// TIA Portal V17 export
// export: Created 2025-04-22T12:08:34.2045134Z, ExportSetting WithDefaults, DisplayName Totally Integrated Automation Portal, DisplayVersion V17 Update 8, DisplayName TIA Portal Openness, DisplayVersion V17 Update 8, DisplayName TIA Portal Version Control Interface, DisplayVersion V17, DisplayName SINAMICS Startdrive Advanced, DisplayVersion V17 SP2, DisplayName SINAMICS Startdrive G110M, G120, G120C, G120D, G120P, G115D, DisplayVersion V17 SP2, DisplayName SINAMICS Startdrive G130, G150, S120, S150, SINAMICS MV, S210, DisplayVersion V17 SP2, DisplayName STEP 7 Professional, DisplayVersion V17 Update 8, DisplayName SINUMERIK ONE STEP 7 Toolbox, DisplayVersion V17 Update 12, DisplayName SINUMERIK 840D sl STEP 7 Toolbox, DisplayVersion V17 Update 12, DisplayName STEP 7 Safety, DisplayVersion V17 Update 6, DisplayName WinCC Advanced / Unified PC, DisplayVersion V17 Update 8
FUNCTION "FC2401_DBBS_CLADDING" : Void   // FC2401, LAD
TITLE = NCK Inputs
{ S7_Optimized_Access := 'FALSE' }
AUTHOR : ETXETAR
VERSION : 1.0
// stored: AutoNumber false, IsIECCheckEnabled false, SetENOAutomatically false, UDAEnableTagReadback false
   VAR_TEMP
      ERROR : Bool;   // ERROR
      ERROR_CODE : Int;   // ERROR CODE
      F1_RESET_SEMI_WORKS : Bool;   // FIXTURE 1 RESET SEMI WORKS
      F2_RESET_SEMI_WORKS : Bool;   // FIXTURE 2 RESET SEMI WORKS
      RESET_UGUD : Bool;   // RESET UGUD
      TAG_ERROR_01R : Int;   // TAG ERROR 01R
      TAG_ERROR_01L : Int;   // TAG ERROR 01L
   END_VAR
   VAR CONSTANT
      READ : Byte := 16#3;
      WRITE : Byte := 16#4;
   END_VAR
BEGIN

REGION Network 1: MACHINE CNC CYCLE UNIT 01 TRANSFER CHANNEL 1 - $A_DBB[0] / CYCLE SELECTION 01R
   // 0 --> NA
   // 1 --> PART CYCLE 01R
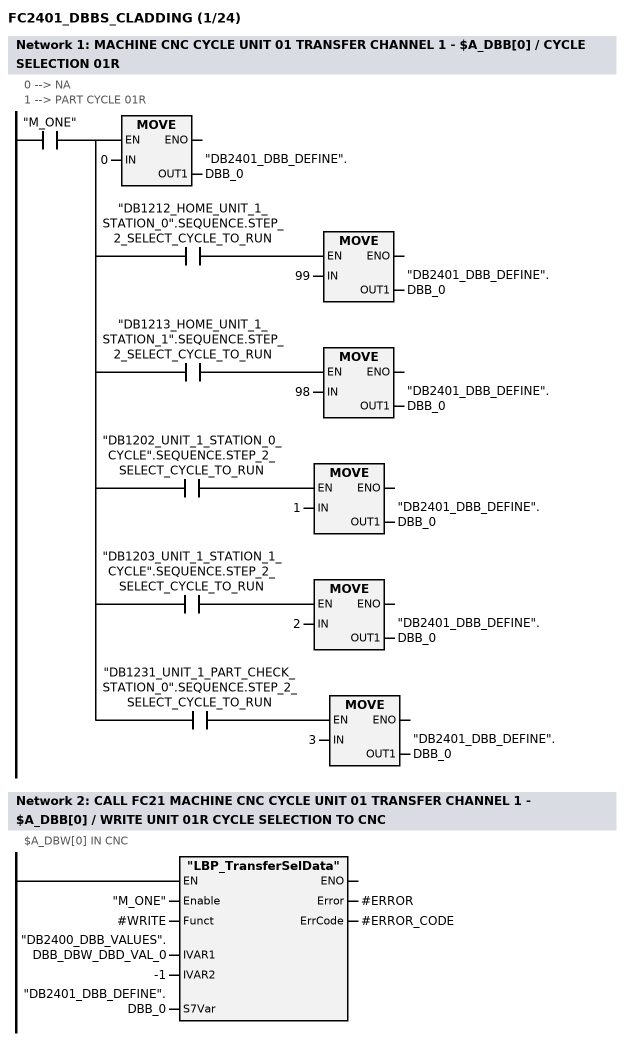
   RUNG wire#powerrail
      Contact( "M_ONE" )
      wire#w1
      { S7_GenerateENO := "TRUE" } Move(in := 0, out1 => "DB2401_DBB_DEFINE".DBB_0)
   END_RUNG
   RUNG wire#w1
      Contact( "DB1212_HOME_UNIT_1_STATION_0".SEQUENCE.STEP_2_SELECT_CYCLE_TO_RUN )
      { S7_GenerateENO := "TRUE" } Move(in := 99, out1 => "DB2401_DBB_DEFINE".DBB_0)
   END_RUNG
   RUNG wire#w1
      Contact( "DB1213_HOME_UNIT_1_STATION_1".SEQUENCE.STEP_2_SELECT_CYCLE_TO_RUN )
      { S7_GenerateENO := "TRUE" } Move(in := 98, out1 => "DB2401_DBB_DEFINE".DBB_0)
   END_RUNG
   RUNG wire#w1
      Contact( "DB1202_UNIT_1_STATION_0_CYCLE".SEQUENCE.STEP_2_SELECT_CYCLE_TO_RUN )
      { S7_GenerateENO := "TRUE" } Move(in := 1, out1 => "DB2401_DBB_DEFINE".DBB_0)
   END_RUNG
   RUNG wire#w1
      Contact( "DB1203_UNIT_1_STATION_1_CYCLE".SEQUENCE.STEP_2_SELECT_CYCLE_TO_RUN )
      { S7_GenerateENO := "TRUE" } Move(in := 2, out1 => "DB2401_DBB_DEFINE".DBB_0)
   END_RUNG
   RUNG wire#w1
      Contact( "DB1231_UNIT_1_PART_CHECK_STATION_0".SEQUENCE.STEP_2_SELECT_CYCLE_TO_RUN )
      { S7_GenerateENO := "TRUE" } Move(in := 3, out1 => "DB2401_DBB_DEFINE".DBB_0)
   END_RUNG
   // the same network as SCL:
   IF "M_ONE" THEN "DB2401_DBB_DEFINE".DBB_0 := 0; END_IF;
   IF "M_ONE" AND "DB1212_HOME_UNIT_1_STATION_0".SEQUENCE.STEP_2_SELECT_CYCLE_TO_RUN THEN
       "DB2401_DBB_DEFINE".DBB_0 := 99;
   END_IF;
   IF "M_ONE" AND "DB1213_HOME_UNIT_1_STATION_1".SEQUENCE.STEP_2_SELECT_CYCLE_TO_RUN THEN
       "DB2401_DBB_DEFINE".DBB_0 := 98;
   END_IF;
   IF "M_ONE" AND "DB1202_UNIT_1_STATION_0_CYCLE".SEQUENCE.STEP_2_SELECT_CYCLE_TO_RUN THEN
       "DB2401_DBB_DEFINE".DBB_0 := 1;
   END_IF;
   IF "M_ONE" AND "DB1203_UNIT_1_STATION_1_CYCLE".SEQUENCE.STEP_2_SELECT_CYCLE_TO_RUN THEN
       "DB2401_DBB_DEFINE".DBB_0 := 2;
   END_IF;
   IF "M_ONE" AND "DB1231_UNIT_1_PART_CHECK_STATION_0".SEQUENCE.STEP_2_SELECT_CYCLE_TO_RUN THEN
       "DB2401_DBB_DEFINE".DBB_0 := 3;
   END_IF;
END_REGION

REGION Network 2: CALL FC21 MACHINE CNC CYCLE UNIT 01 TRANSFER CHANNEL 1 - $A_DBB[0] / WRITE UNIT 01R CYCLE SELECTION TO CNC
   // $A_DBW[0] IN CNC
   RUNG wire#powerrail
      "LBP_TransferSelData"(Enable := "M_ONE", Funct := #WRITE, IVAR1 := "DB2400_DBB_VALUES".DBB_DBW_DBD_VAL_0, IVAR2 := -1, S7Var := "DB2401_DBB_DEFINE".DBB_0, Error => #ERROR, ErrCode => #ERROR_CODE)
   END_RUNG
   // the same network as SCL:
   "LBP_TransferSelData"(Enable := "M_ONE",
                         Funct := #WRITE,
                         IVAR1 := "DB2400_DBB_VALUES".DBB_DBW_DBD_VAL_0,
                         IVAR2 := -1,
                         S7Var := "DB2401_DBB_DEFINE".DBB_0,
                         Error => #ERROR,
                         ErrCode => #ERROR_CODE);
END_REGION

REGION Network 3: MACHINE CNC CYCLE UNIT 01 CLADDING CHANNEL 2 - $A_DBB[2] / CYCLE SELECTION PHD
   // 0 --> NA
   // 1 --> PHD CYCLE
   // 99 --> RETURN HOME CYCLE PHD
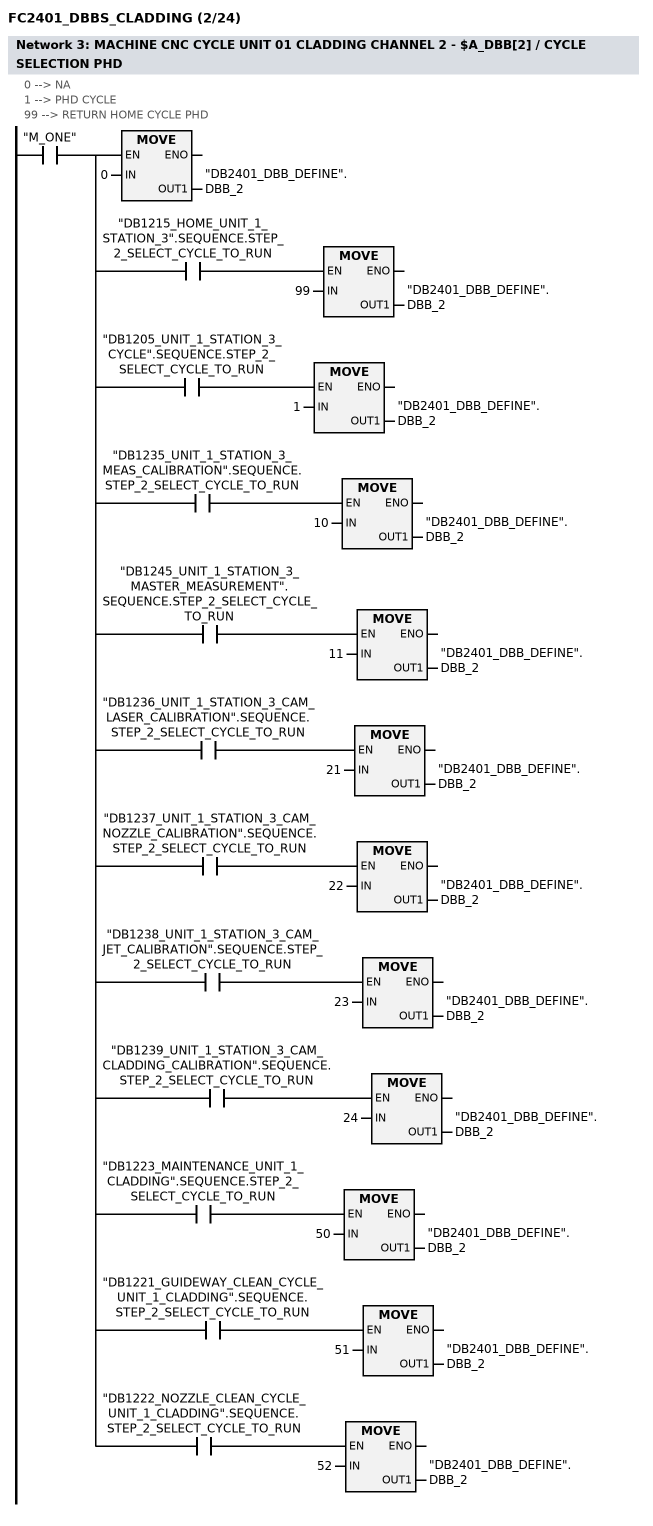
   RUNG wire#powerrail
      Contact( "M_ONE" )
      wire#w1
      { S7_GenerateENO := "TRUE" } Move(in := 0, out1 => "DB2401_DBB_DEFINE".DBB_2)
   END_RUNG
   RUNG wire#w1
      Contact( "DB1215_HOME_UNIT_1_STATION_3".SEQUENCE.STEP_2_SELECT_CYCLE_TO_RUN )
      { S7_GenerateENO := "TRUE" } Move(in := 99, out1 => "DB2401_DBB_DEFINE".DBB_2)
   END_RUNG
   RUNG wire#w1
      Contact( "DB1205_UNIT_1_STATION_3_CYCLE".SEQUENCE.STEP_2_SELECT_CYCLE_TO_RUN )
      { S7_GenerateENO := "TRUE" } Move(in := 1, out1 => "DB2401_DBB_DEFINE".DBB_2)
   END_RUNG
   RUNG wire#w1
      Contact( "DB1235_UNIT_1_STATION_3_MEAS_CALIBRATION".SEQUENCE.STEP_2_SELECT_CYCLE_TO_RUN )
      { S7_GenerateENO := "TRUE" } Move(in := 10, out1 => "DB2401_DBB_DEFINE".DBB_2)
   END_RUNG
   RUNG wire#w1
      Contact( "DB1245_UNIT_1_STATION_3_MASTER_MEASUREMENT".SEQUENCE.STEP_2_SELECT_CYCLE_TO_RUN )
      { S7_GenerateENO := "TRUE" } Move(in := 11, out1 => "DB2401_DBB_DEFINE".DBB_2)
   END_RUNG
   RUNG wire#w1
      Contact( "DB1236_UNIT_1_STATION_3_CAM_LASER_CALIBRATION".SEQUENCE.STEP_2_SELECT_CYCLE_TO_RUN )
      { S7_GenerateENO := "TRUE" } Move(in := 21, out1 => "DB2401_DBB_DEFINE".DBB_2)
   END_RUNG
   RUNG wire#w1
      Contact( "DB1237_UNIT_1_STATION_3_CAM_NOZZLE_CALIBRATION".SEQUENCE.STEP_2_SELECT_CYCLE_TO_RUN )
      { S7_GenerateENO := "TRUE" } Move(in := 22, out1 => "DB2401_DBB_DEFINE".DBB_2)
   END_RUNG
   RUNG wire#w1
      Contact( "DB1238_UNIT_1_STATION_3_CAM_JET_CALIBRATION".SEQUENCE.STEP_2_SELECT_CYCLE_TO_RUN )
      { S7_GenerateENO := "TRUE" } Move(in := 23, out1 => "DB2401_DBB_DEFINE".DBB_2)
   END_RUNG
   RUNG wire#w1
      Contact( "DB1239_UNIT_1_STATION_3_CAM_CLADDING_CALIBRATION".SEQUENCE.STEP_2_SELECT_CYCLE_TO_RUN )
      { S7_GenerateENO := "TRUE" } Move(in := 24, out1 => "DB2401_DBB_DEFINE".DBB_2)
   END_RUNG
   RUNG wire#w1
      Contact( "DB1223_MAINTENANCE_UNIT_1_CLADDING".SEQUENCE.STEP_2_SELECT_CYCLE_TO_RUN )
      { S7_GenerateENO := "TRUE" } Move(in := 50, out1 => "DB2401_DBB_DEFINE".DBB_2)
   END_RUNG
   RUNG wire#w1
      Contact( "DB1221_GUIDEWAY_CLEAN_CYCLE_UNIT_1_CLADDING".SEQUENCE.STEP_2_SELECT_CYCLE_TO_RUN )
      { S7_GenerateENO := "TRUE" } Move(in := 51, out1 => "DB2401_DBB_DEFINE".DBB_2)
   END_RUNG
   RUNG wire#w1
      Contact( "DB1222_NOZZLE_CLEAN_CYCLE_UNIT_1_CLADDING".SEQUENCE.STEP_2_SELECT_CYCLE_TO_RUN )
      { S7_GenerateENO := "TRUE" } Move(in := 52, out1 => "DB2401_DBB_DEFINE".DBB_2)
   END_RUNG
   // the same network as SCL:
   IF "M_ONE" THEN "DB2401_DBB_DEFINE".DBB_2 := 0; END_IF;
   IF "M_ONE" AND "DB1215_HOME_UNIT_1_STATION_3".SEQUENCE.STEP_2_SELECT_CYCLE_TO_RUN THEN
       "DB2401_DBB_DEFINE".DBB_2 := 99;
   END_IF;
   IF "M_ONE" AND "DB1205_UNIT_1_STATION_3_CYCLE".SEQUENCE.STEP_2_SELECT_CYCLE_TO_RUN THEN
       "DB2401_DBB_DEFINE".DBB_2 := 1;
   END_IF;
   IF "M_ONE" AND "DB1235_UNIT_1_STATION_3_MEAS_CALIBRATION".SEQUENCE.STEP_2_SELECT_CYCLE_TO_RUN THEN
       "DB2401_DBB_DEFINE".DBB_2 := 10;
   END_IF;
   IF "M_ONE" AND "DB1245_UNIT_1_STATION_3_MASTER_MEASUREMENT".SEQUENCE.STEP_2_SELECT_CYCLE_TO_RUN THEN
       "DB2401_DBB_DEFINE".DBB_2 := 11;
   END_IF;
   IF "M_ONE" AND "DB1236_UNIT_1_STATION_3_CAM_LASER_CALIBRATION".SEQUENCE.STEP_2_SELECT_CYCLE_TO_RUN THEN
       "DB2401_DBB_DEFINE".DBB_2 := 21;
   END_IF;
   IF "M_ONE" AND "DB1237_UNIT_1_STATION_3_CAM_NOZZLE_CALIBRATION".SEQUENCE.STEP_2_SELECT_CYCLE_TO_RUN THEN
       "DB2401_DBB_DEFINE".DBB_2 := 22;
   END_IF;
   IF "M_ONE" AND "DB1238_UNIT_1_STATION_3_CAM_JET_CALIBRATION".SEQUENCE.STEP_2_SELECT_CYCLE_TO_RUN THEN
       "DB2401_DBB_DEFINE".DBB_2 := 23;
   END_IF;
   IF "M_ONE" AND "DB1239_UNIT_1_STATION_3_CAM_CLADDING_CALIBRATION".SEQUENCE.STEP_2_SELECT_CYCLE_TO_RUN THEN
       "DB2401_DBB_DEFINE".DBB_2 := 24;
   END_IF;
   IF "M_ONE" AND "DB1223_MAINTENANCE_UNIT_1_CLADDING".SEQUENCE.STEP_2_SELECT_CYCLE_TO_RUN THEN
       "DB2401_DBB_DEFINE".DBB_2 := 50;
   END_IF;
   IF "M_ONE" AND "DB1221_GUIDEWAY_CLEAN_CYCLE_UNIT_1_CLADDING".SEQUENCE.STEP_2_SELECT_CYCLE_TO_RUN THEN
       "DB2401_DBB_DEFINE".DBB_2 := 51;
   END_IF;
   IF "M_ONE" AND "DB1222_NOZZLE_CLEAN_CYCLE_UNIT_1_CLADDING".SEQUENCE.STEP_2_SELECT_CYCLE_TO_RUN THEN
       "DB2401_DBB_DEFINE".DBB_2 := 52;
   END_IF;
END_REGION

REGION Network 4: CALL FC21 MACHINE CNC CYCLE UNIT 01 CLADDING CHANNEL 2 - $A_DBB[2] / WRITE UNIT 01R CYCLE SELECTION TO CNC
   // $A_DBW[0] IN CNC
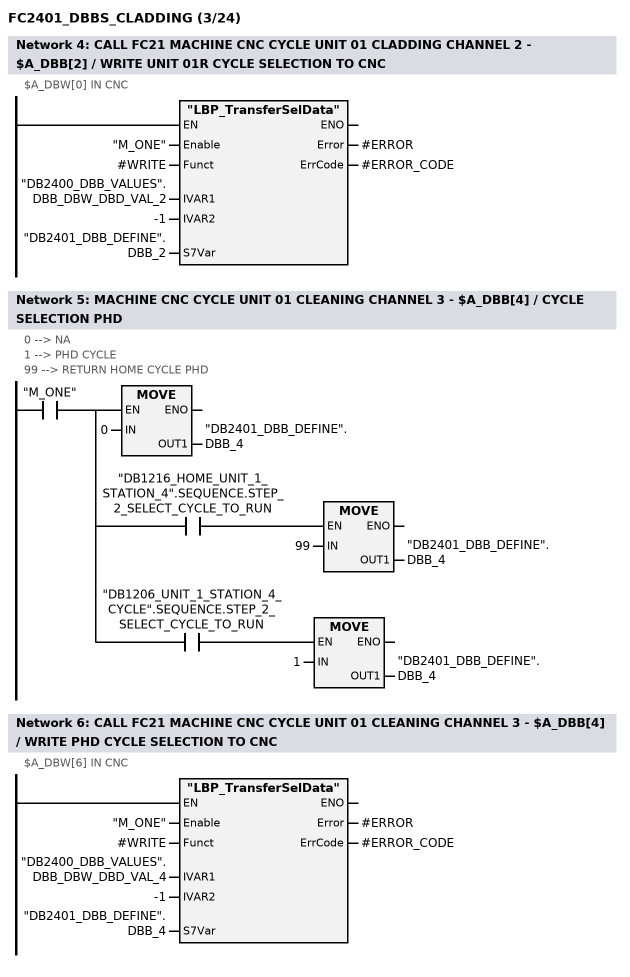
   RUNG wire#powerrail
      "LBP_TransferSelData"(Enable := "M_ONE", Funct := #WRITE, IVAR1 := "DB2400_DBB_VALUES".DBB_DBW_DBD_VAL_2, IVAR2 := -1, S7Var := "DB2401_DBB_DEFINE".DBB_2, Error => #ERROR, ErrCode => #ERROR_CODE)
   END_RUNG
   // the same network as SCL:
   "LBP_TransferSelData"(Enable := "M_ONE",
                         Funct := #WRITE,
                         IVAR1 := "DB2400_DBB_VALUES".DBB_DBW_DBD_VAL_2,
                         IVAR2 := -1,
                         S7Var := "DB2401_DBB_DEFINE".DBB_2,
                         Error => #ERROR,
                         ErrCode => #ERROR_CODE);
END_REGION

REGION Network 5: MACHINE CNC CYCLE UNIT 01 CLEANING CHANNEL 3 - $A_DBB[4] / CYCLE SELECTION PHD
   // 0 --> NA
   // 1 --> PHD CYCLE
   // 99 --> RETURN HOME CYCLE PHD
   RUNG wire#powerrail
      Contact( "M_ONE" )
      wire#w1
      { S7_GenerateENO := "TRUE" } Move(in := 0, out1 => "DB2401_DBB_DEFINE".DBB_4)
   END_RUNG
   RUNG wire#w1
      Contact( "DB1216_HOME_UNIT_1_STATION_4".SEQUENCE.STEP_2_SELECT_CYCLE_TO_RUN )
      { S7_GenerateENO := "TRUE" } Move(in := 99, out1 => "DB2401_DBB_DEFINE".DBB_4)
   END_RUNG
   RUNG wire#w1
      Contact( "DB1206_UNIT_1_STATION_4_CYCLE".SEQUENCE.STEP_2_SELECT_CYCLE_TO_RUN )
      { S7_GenerateENO := "TRUE" } Move(in := 1, out1 => "DB2401_DBB_DEFINE".DBB_4)
   END_RUNG
   // the same network as SCL:
   IF "M_ONE" THEN "DB2401_DBB_DEFINE".DBB_4 := 0; END_IF;
   IF "M_ONE" AND "DB1216_HOME_UNIT_1_STATION_4".SEQUENCE.STEP_2_SELECT_CYCLE_TO_RUN THEN
       "DB2401_DBB_DEFINE".DBB_4 := 99;
   END_IF;
   IF "M_ONE" AND "DB1206_UNIT_1_STATION_4_CYCLE".SEQUENCE.STEP_2_SELECT_CYCLE_TO_RUN THEN
       "DB2401_DBB_DEFINE".DBB_4 := 1;
   END_IF;
END_REGION

REGION Network 6: CALL FC21 MACHINE CNC CYCLE UNIT 01 CLEANING CHANNEL 3 - $A_DBB[4] / WRITE PHD CYCLE SELECTION TO CNC
   // $A_DBW[6] IN CNC
   RUNG wire#powerrail
      "LBP_TransferSelData"(Enable := "M_ONE", Funct := #WRITE, IVAR1 := "DB2400_DBB_VALUES".DBB_DBW_DBD_VAL_4, IVAR2 := -1, S7Var := "DB2401_DBB_DEFINE".DBB_4, Error => #ERROR, ErrCode => #ERROR_CODE)
   END_RUNG
   // the same network as SCL:
   "LBP_TransferSelData"(Enable := "M_ONE",
                         Funct := #WRITE,
                         IVAR1 := "DB2400_DBB_VALUES".DBB_DBW_DBD_VAL_4,
                         IVAR2 := -1,
                         S7Var := "DB2401_DBB_DEFINE".DBB_4,
                         Error => #ERROR,
                         ErrCode => #ERROR_CODE);
END_REGION

REGION Network 7: MACHINE CNC CYCLE UNIT 02 TRANSFER CHANNEL 4 - $A_DBB[6] / CYCLE SELECTION PHD
   // 0 --> NA
   // 1 --> PHD CYCLE
   // 99 --> RETURN HOME CYCLE PHD
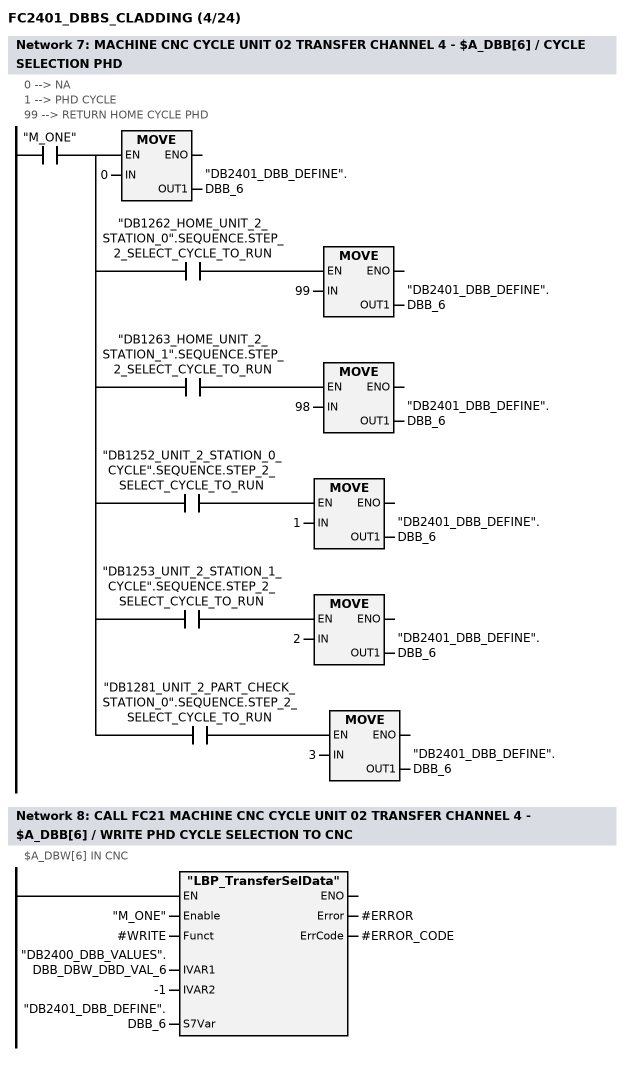
   RUNG wire#powerrail
      Contact( "M_ONE" )
      wire#w1
      { S7_GenerateENO := "TRUE" } Move(in := 0, out1 => "DB2401_DBB_DEFINE".DBB_6)
   END_RUNG
   RUNG wire#w1
      Contact( "DB1262_HOME_UNIT_2_STATION_0".SEQUENCE.STEP_2_SELECT_CYCLE_TO_RUN )
      { S7_GenerateENO := "TRUE" } Move(in := 99, out1 => "DB2401_DBB_DEFINE".DBB_6)
   END_RUNG
   RUNG wire#w1
      Contact( "DB1263_HOME_UNIT_2_STATION_1".SEQUENCE.STEP_2_SELECT_CYCLE_TO_RUN )
      { S7_GenerateENO := "TRUE" } Move(in := 98, out1 => "DB2401_DBB_DEFINE".DBB_6)
   END_RUNG
   RUNG wire#w1
      Contact( "DB1252_UNIT_2_STATION_0_CYCLE".SEQUENCE.STEP_2_SELECT_CYCLE_TO_RUN )
      { S7_GenerateENO := "TRUE" } Move(in := 1, out1 => "DB2401_DBB_DEFINE".DBB_6)
   END_RUNG
   RUNG wire#w1
      Contact( "DB1253_UNIT_2_STATION_1_CYCLE".SEQUENCE.STEP_2_SELECT_CYCLE_TO_RUN )
      { S7_GenerateENO := "TRUE" } Move(in := 2, out1 => "DB2401_DBB_DEFINE".DBB_6)
   END_RUNG
   RUNG wire#w1
      Contact( "DB1281_UNIT_2_PART_CHECK_STATION_0".SEQUENCE.STEP_2_SELECT_CYCLE_TO_RUN )
      { S7_GenerateENO := "TRUE" } Move(in := 3, out1 => "DB2401_DBB_DEFINE".DBB_6)
   END_RUNG
   // the same network as SCL:
   IF "M_ONE" THEN "DB2401_DBB_DEFINE".DBB_6 := 0; END_IF;
   IF "M_ONE" AND "DB1262_HOME_UNIT_2_STATION_0".SEQUENCE.STEP_2_SELECT_CYCLE_TO_RUN THEN
       "DB2401_DBB_DEFINE".DBB_6 := 99;
   END_IF;
   IF "M_ONE" AND "DB1263_HOME_UNIT_2_STATION_1".SEQUENCE.STEP_2_SELECT_CYCLE_TO_RUN THEN
       "DB2401_DBB_DEFINE".DBB_6 := 98;
   END_IF;
   IF "M_ONE" AND "DB1252_UNIT_2_STATION_0_CYCLE".SEQUENCE.STEP_2_SELECT_CYCLE_TO_RUN THEN
       "DB2401_DBB_DEFINE".DBB_6 := 1;
   END_IF;
   IF "M_ONE" AND "DB1253_UNIT_2_STATION_1_CYCLE".SEQUENCE.STEP_2_SELECT_CYCLE_TO_RUN THEN
       "DB2401_DBB_DEFINE".DBB_6 := 2;
   END_IF;
   IF "M_ONE" AND "DB1281_UNIT_2_PART_CHECK_STATION_0".SEQUENCE.STEP_2_SELECT_CYCLE_TO_RUN THEN
       "DB2401_DBB_DEFINE".DBB_6 := 3;
   END_IF;
END_REGION

REGION Network 8: CALL FC21 MACHINE CNC CYCLE UNIT 02 TRANSFER CHANNEL 4 - $A_DBB[6] / WRITE PHD CYCLE SELECTION TO CNC
   // $A_DBW[6] IN CNC
   RUNG wire#powerrail
      "LBP_TransferSelData"(Enable := "M_ONE", Funct := #WRITE, IVAR1 := "DB2400_DBB_VALUES".DBB_DBW_DBD_VAL_6, IVAR2 := -1, S7Var := "DB2401_DBB_DEFINE".DBB_6, Error => #ERROR, ErrCode => #ERROR_CODE)
   END_RUNG
   // the same network as SCL:
   "LBP_TransferSelData"(Enable := "M_ONE",
                         Funct := #WRITE,
                         IVAR1 := "DB2400_DBB_VALUES".DBB_DBW_DBD_VAL_6,
                         IVAR2 := -1,
                         S7Var := "DB2401_DBB_DEFINE".DBB_6,
                         Error => #ERROR,
                         ErrCode => #ERROR_CODE);
END_REGION

REGION Network 9: MACHINE CNC CYCLE UNIT 02 MEASURING CHANNEL 5 - $A_DBB[8] / CYCLE SELECTION PHD
   // 0 --> NA
   // 1 --> PHD CYCLE
   // 99 --> RETURN HOME CYCLE PHD
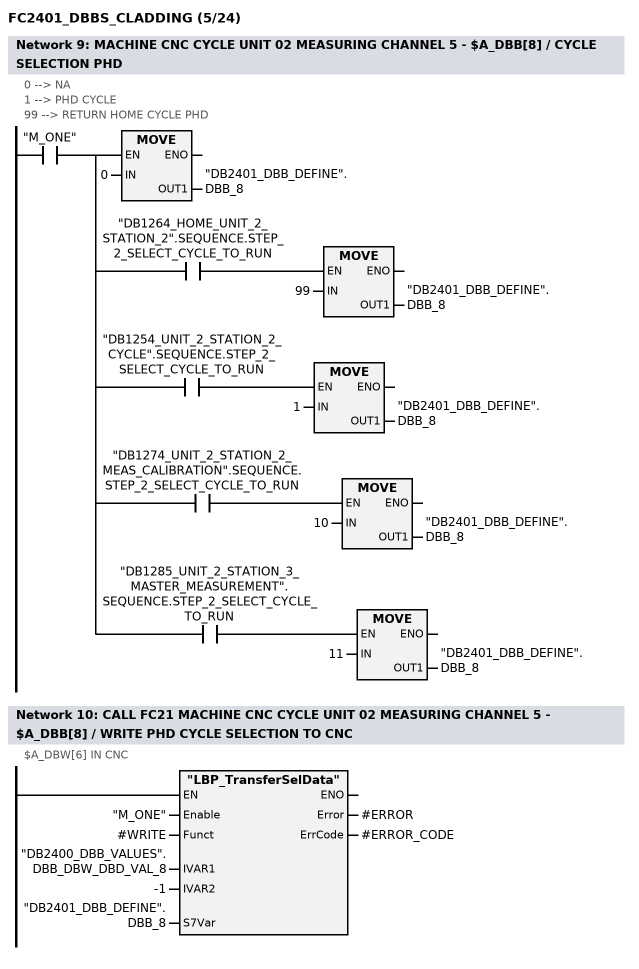
   RUNG wire#powerrail
      Contact( "M_ONE" )
      wire#w1
      { S7_GenerateENO := "TRUE" } Move(in := 0, out1 => "DB2401_DBB_DEFINE".DBB_8)
   END_RUNG
   RUNG wire#w1
      Contact( "DB1264_HOME_UNIT_2_STATION_2".SEQUENCE.STEP_2_SELECT_CYCLE_TO_RUN )
      { S7_GenerateENO := "TRUE" } Move(in := 99, out1 => "DB2401_DBB_DEFINE".DBB_8)
   END_RUNG
   RUNG wire#w1
      Contact( "DB1254_UNIT_2_STATION_2_CYCLE".SEQUENCE.STEP_2_SELECT_CYCLE_TO_RUN )
      { S7_GenerateENO := "TRUE" } Move(in := 1, out1 => "DB2401_DBB_DEFINE".DBB_8)
   END_RUNG
   RUNG wire#w1
      Contact( "DB1274_UNIT_2_STATION_2_MEAS_CALIBRATION".SEQUENCE.STEP_2_SELECT_CYCLE_TO_RUN )
      { S7_GenerateENO := "TRUE" } Move(in := 10, out1 => "DB2401_DBB_DEFINE".DBB_8)
   END_RUNG
   RUNG wire#w1
      Contact( "DB1285_UNIT_2_STATION_3_MASTER_MEASUREMENT".SEQUENCE.STEP_2_SELECT_CYCLE_TO_RUN )
      { S7_GenerateENO := "TRUE" } Move(in := 11, out1 => "DB2401_DBB_DEFINE".DBB_8)
   END_RUNG
   // the same network as SCL:
   IF "M_ONE" THEN "DB2401_DBB_DEFINE".DBB_8 := 0; END_IF;
   IF "M_ONE" AND "DB1264_HOME_UNIT_2_STATION_2".SEQUENCE.STEP_2_SELECT_CYCLE_TO_RUN THEN
       "DB2401_DBB_DEFINE".DBB_8 := 99;
   END_IF;
   IF "M_ONE" AND "DB1254_UNIT_2_STATION_2_CYCLE".SEQUENCE.STEP_2_SELECT_CYCLE_TO_RUN THEN
       "DB2401_DBB_DEFINE".DBB_8 := 1;
   END_IF;
   IF "M_ONE" AND "DB1274_UNIT_2_STATION_2_MEAS_CALIBRATION".SEQUENCE.STEP_2_SELECT_CYCLE_TO_RUN THEN
       "DB2401_DBB_DEFINE".DBB_8 := 10;
   END_IF;
   IF "M_ONE" AND "DB1285_UNIT_2_STATION_3_MASTER_MEASUREMENT".SEQUENCE.STEP_2_SELECT_CYCLE_TO_RUN THEN
       "DB2401_DBB_DEFINE".DBB_8 := 11;
   END_IF;
END_REGION

REGION Network 10: CALL FC21 MACHINE CNC CYCLE UNIT 02 MEASURING CHANNEL 5 - $A_DBB[8] / WRITE PHD CYCLE SELECTION TO CNC
   // $A_DBW[6] IN CNC
   RUNG wire#powerrail
      "LBP_TransferSelData"(Enable := "M_ONE", Funct := #WRITE, IVAR1 := "DB2400_DBB_VALUES".DBB_DBW_DBD_VAL_8, IVAR2 := -1, S7Var := "DB2401_DBB_DEFINE".DBB_8, Error => #ERROR, ErrCode => #ERROR_CODE)
   END_RUNG
   // the same network as SCL:
   "LBP_TransferSelData"(Enable := "M_ONE",
                         Funct := #WRITE,
                         IVAR1 := "DB2400_DBB_VALUES".DBB_DBW_DBD_VAL_8,
                         IVAR2 := -1,
                         S7Var := "DB2401_DBB_DEFINE".DBB_8,
                         Error => #ERROR,
                         ErrCode => #ERROR_CODE);
END_REGION

REGION Network 11: MACHINE CNC CYCLE UNIT 02 CLADDING CHANNEL 6 - $A_DBB[10] / CYCLE SELECTION PHD
   // 0 --> NA
   // 1 --> PHD CYCLE
   // 99 --> RETURN HOME CYCLE PHD
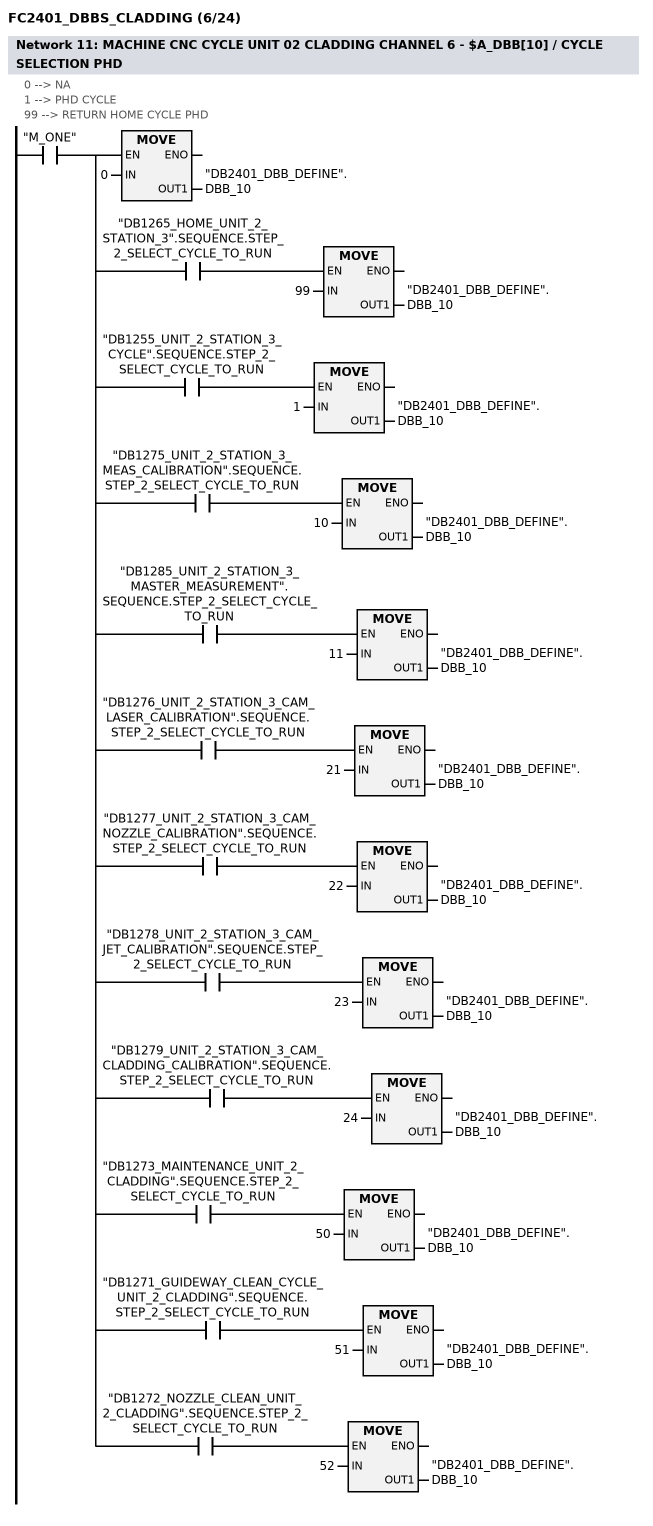
   RUNG wire#powerrail
      Contact( "M_ONE" )
      wire#w1
      { S7_GenerateENO := "TRUE" } Move(in := 0, out1 => "DB2401_DBB_DEFINE".DBB_10)
   END_RUNG
   RUNG wire#w1
      Contact( "DB1265_HOME_UNIT_2_STATION_3".SEQUENCE.STEP_2_SELECT_CYCLE_TO_RUN )
      { S7_GenerateENO := "TRUE" } Move(in := 99, out1 => "DB2401_DBB_DEFINE".DBB_10)
   END_RUNG
   RUNG wire#w1
      Contact( "DB1255_UNIT_2_STATION_3_CYCLE".SEQUENCE.STEP_2_SELECT_CYCLE_TO_RUN )
      { S7_GenerateENO := "TRUE" } Move(in := 1, out1 => "DB2401_DBB_DEFINE".DBB_10)
   END_RUNG
   RUNG wire#w1
      Contact( "DB1275_UNIT_2_STATION_3_MEAS_CALIBRATION".SEQUENCE.STEP_2_SELECT_CYCLE_TO_RUN )
      { S7_GenerateENO := "TRUE" } Move(in := 10, out1 => "DB2401_DBB_DEFINE".DBB_10)
   END_RUNG
   RUNG wire#w1
      Contact( "DB1285_UNIT_2_STATION_3_MASTER_MEASUREMENT".SEQUENCE.STEP_2_SELECT_CYCLE_TO_RUN )
      { S7_GenerateENO := "TRUE" } Move(in := 11, out1 => "DB2401_DBB_DEFINE".DBB_10)
   END_RUNG
   RUNG wire#w1
      Contact( "DB1276_UNIT_2_STATION_3_CAM_LASER_CALIBRATION".SEQUENCE.STEP_2_SELECT_CYCLE_TO_RUN )
      { S7_GenerateENO := "TRUE" } Move(in := 21, out1 => "DB2401_DBB_DEFINE".DBB_10)
   END_RUNG
   RUNG wire#w1
      Contact( "DB1277_UNIT_2_STATION_3_CAM_NOZZLE_CALIBRATION".SEQUENCE.STEP_2_SELECT_CYCLE_TO_RUN )
      { S7_GenerateENO := "TRUE" } Move(in := 22, out1 => "DB2401_DBB_DEFINE".DBB_10)
   END_RUNG
   RUNG wire#w1
      Contact( "DB1278_UNIT_2_STATION_3_CAM_JET_CALIBRATION".SEQUENCE.STEP_2_SELECT_CYCLE_TO_RUN )
      { S7_GenerateENO := "TRUE" } Move(in := 23, out1 => "DB2401_DBB_DEFINE".DBB_10)
   END_RUNG
   RUNG wire#w1
      Contact( "DB1279_UNIT_2_STATION_3_CAM_CLADDING_CALIBRATION".SEQUENCE.STEP_2_SELECT_CYCLE_TO_RUN )
      { S7_GenerateENO := "TRUE" } Move(in := 24, out1 => "DB2401_DBB_DEFINE".DBB_10)
   END_RUNG
   RUNG wire#w1
      Contact( "DB1273_MAINTENANCE_UNIT_2_CLADDING".SEQUENCE.STEP_2_SELECT_CYCLE_TO_RUN )
      { S7_GenerateENO := "TRUE" } Move(in := 50, out1 => "DB2401_DBB_DEFINE".DBB_10)
   END_RUNG
   RUNG wire#w1
      Contact( "DB1271_GUIDEWAY_CLEAN_CYCLE_UNIT_2_CLADDING".SEQUENCE.STEP_2_SELECT_CYCLE_TO_RUN )
      { S7_GenerateENO := "TRUE" } Move(in := 51, out1 => "DB2401_DBB_DEFINE".DBB_10)
   END_RUNG
   RUNG wire#w1
      Contact( "DB1272_NOZZLE_CLEAN_UNIT_2_CLADDING".SEQUENCE.STEP_2_SELECT_CYCLE_TO_RUN )
      { S7_GenerateENO := "TRUE" } Move(in := 52, out1 => "DB2401_DBB_DEFINE".DBB_10)
   END_RUNG
   // the same network as SCL:
   IF "M_ONE" THEN "DB2401_DBB_DEFINE".DBB_10 := 0; END_IF;
   IF "M_ONE" AND "DB1265_HOME_UNIT_2_STATION_3".SEQUENCE.STEP_2_SELECT_CYCLE_TO_RUN THEN
       "DB2401_DBB_DEFINE".DBB_10 := 99;
   END_IF;
   IF "M_ONE" AND "DB1255_UNIT_2_STATION_3_CYCLE".SEQUENCE.STEP_2_SELECT_CYCLE_TO_RUN THEN
       "DB2401_DBB_DEFINE".DBB_10 := 1;
   END_IF;
   IF "M_ONE" AND "DB1275_UNIT_2_STATION_3_MEAS_CALIBRATION".SEQUENCE.STEP_2_SELECT_CYCLE_TO_RUN THEN
       "DB2401_DBB_DEFINE".DBB_10 := 10;
   END_IF;
   IF "M_ONE" AND "DB1285_UNIT_2_STATION_3_MASTER_MEASUREMENT".SEQUENCE.STEP_2_SELECT_CYCLE_TO_RUN THEN
       "DB2401_DBB_DEFINE".DBB_10 := 11;
   END_IF;
   IF "M_ONE" AND "DB1276_UNIT_2_STATION_3_CAM_LASER_CALIBRATION".SEQUENCE.STEP_2_SELECT_CYCLE_TO_RUN THEN
       "DB2401_DBB_DEFINE".DBB_10 := 21;
   END_IF;
   IF "M_ONE" AND "DB1277_UNIT_2_STATION_3_CAM_NOZZLE_CALIBRATION".SEQUENCE.STEP_2_SELECT_CYCLE_TO_RUN THEN
       "DB2401_DBB_DEFINE".DBB_10 := 22;
   END_IF;
   IF "M_ONE" AND "DB1278_UNIT_2_STATION_3_CAM_JET_CALIBRATION".SEQUENCE.STEP_2_SELECT_CYCLE_TO_RUN THEN
       "DB2401_DBB_DEFINE".DBB_10 := 23;
   END_IF;
   IF "M_ONE" AND "DB1279_UNIT_2_STATION_3_CAM_CLADDING_CALIBRATION".SEQUENCE.STEP_2_SELECT_CYCLE_TO_RUN THEN
       "DB2401_DBB_DEFINE".DBB_10 := 24;
   END_IF;
   IF "M_ONE" AND "DB1273_MAINTENANCE_UNIT_2_CLADDING".SEQUENCE.STEP_2_SELECT_CYCLE_TO_RUN THEN
       "DB2401_DBB_DEFINE".DBB_10 := 50;
   END_IF;
   IF "M_ONE" AND "DB1271_GUIDEWAY_CLEAN_CYCLE_UNIT_2_CLADDING".SEQUENCE.STEP_2_SELECT_CYCLE_TO_RUN THEN
       "DB2401_DBB_DEFINE".DBB_10 := 51;
   END_IF;
   IF "M_ONE" AND "DB1272_NOZZLE_CLEAN_UNIT_2_CLADDING".SEQUENCE.STEP_2_SELECT_CYCLE_TO_RUN THEN
       "DB2401_DBB_DEFINE".DBB_10 := 52;
   END_IF;
END_REGION

REGION Network 12: CALL FC21 MACHINE CNC CYCLE UNIT 02 CLADDING CHANNEL 6 - $A_DBB[10] / WRITE PHD CYCLE SELECTION TO CNC
   // $A_DBW[6] IN CNC
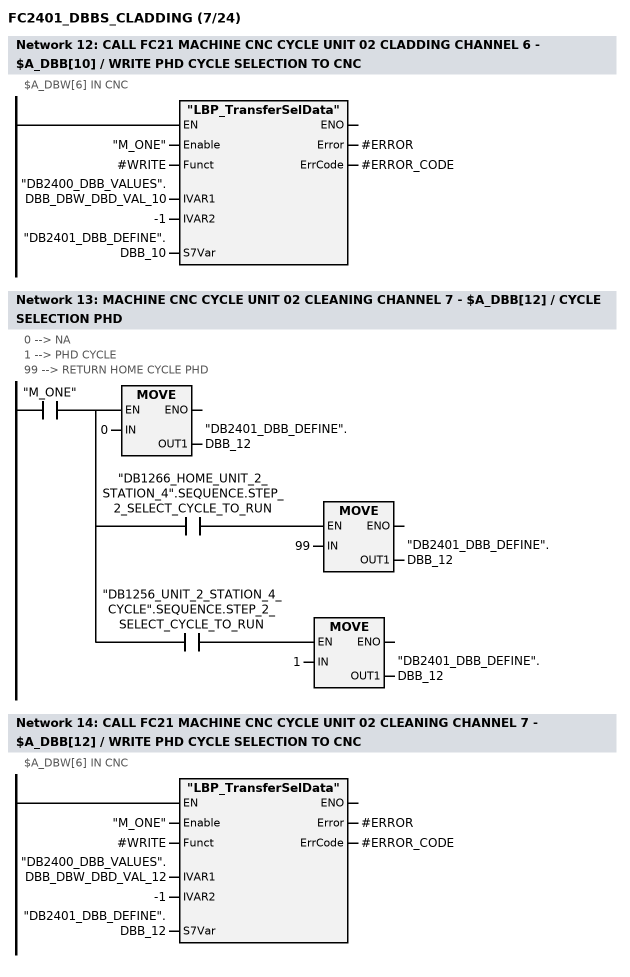
   RUNG wire#powerrail
      "LBP_TransferSelData"(Enable := "M_ONE", Funct := #WRITE, IVAR1 := "DB2400_DBB_VALUES".DBB_DBW_DBD_VAL_10, IVAR2 := -1, S7Var := "DB2401_DBB_DEFINE".DBB_10, Error => #ERROR, ErrCode => #ERROR_CODE)
   END_RUNG
   // the same network as SCL:
   "LBP_TransferSelData"(Enable := "M_ONE",
                         Funct := #WRITE,
                         IVAR1 := "DB2400_DBB_VALUES".DBB_DBW_DBD_VAL_10,
                         IVAR2 := -1,
                         S7Var := "DB2401_DBB_DEFINE".DBB_10,
                         Error => #ERROR,
                         ErrCode => #ERROR_CODE);
END_REGION

REGION Network 13: MACHINE CNC CYCLE UNIT 02 CLEANING CHANNEL 7 - $A_DBB[12] / CYCLE SELECTION PHD
   // 0 --> NA
   // 1 --> PHD CYCLE
   // 99 --> RETURN HOME CYCLE PHD
   RUNG wire#powerrail
      Contact( "M_ONE" )
      wire#w1
      { S7_GenerateENO := "TRUE" } Move(in := 0, out1 => "DB2401_DBB_DEFINE".DBB_12)
   END_RUNG
   RUNG wire#w1
      Contact( "DB1266_HOME_UNIT_2_STATION_4".SEQUENCE.STEP_2_SELECT_CYCLE_TO_RUN )
      { S7_GenerateENO := "TRUE" } Move(in := 99, out1 => "DB2401_DBB_DEFINE".DBB_12)
   END_RUNG
   RUNG wire#w1
      Contact( "DB1256_UNIT_2_STATION_4_CYCLE".SEQUENCE.STEP_2_SELECT_CYCLE_TO_RUN )
      { S7_GenerateENO := "TRUE" } Move(in := 1, out1 => "DB2401_DBB_DEFINE".DBB_12)
   END_RUNG
   // the same network as SCL:
   IF "M_ONE" THEN "DB2401_DBB_DEFINE".DBB_12 := 0; END_IF;
   IF "M_ONE" AND "DB1266_HOME_UNIT_2_STATION_4".SEQUENCE.STEP_2_SELECT_CYCLE_TO_RUN THEN
       "DB2401_DBB_DEFINE".DBB_12 := 99;
   END_IF;
   IF "M_ONE" AND "DB1256_UNIT_2_STATION_4_CYCLE".SEQUENCE.STEP_2_SELECT_CYCLE_TO_RUN THEN
       "DB2401_DBB_DEFINE".DBB_12 := 1;
   END_IF;
END_REGION

REGION Network 14: CALL FC21 MACHINE CNC CYCLE UNIT 02 CLEANING CHANNEL 7 - $A_DBB[12] / WRITE PHD CYCLE SELECTION TO CNC
   // $A_DBW[6] IN CNC
   RUNG wire#powerrail
      "LBP_TransferSelData"(Enable := "M_ONE", Funct := #WRITE, IVAR1 := "DB2400_DBB_VALUES".DBB_DBW_DBD_VAL_12, IVAR2 := -1, S7Var := "DB2401_DBB_DEFINE".DBB_12, Error => #ERROR, ErrCode => #ERROR_CODE)
   END_RUNG
   // the same network as SCL:
   "LBP_TransferSelData"(Enable := "M_ONE",
                         Funct := #WRITE,
                         IVAR1 := "DB2400_DBB_VALUES".DBB_DBW_DBD_VAL_12,
                         IVAR2 := -1,
                         S7Var := "DB2401_DBB_DEFINE".DBB_12,
                         Error => #ERROR,
                         ErrCode => #ERROR_CODE);
END_REGION

REGION Network 15: MACHINE CNC CYCLE UNIT 03 CLEANING CHANNEL 8 - $A_DBB[14] / CYCLE SELECTION PHD
   // 0 --> NA
   // 1 --> PHD CYCLE
   // 99 --> RETURN HOME CYCLE PHD
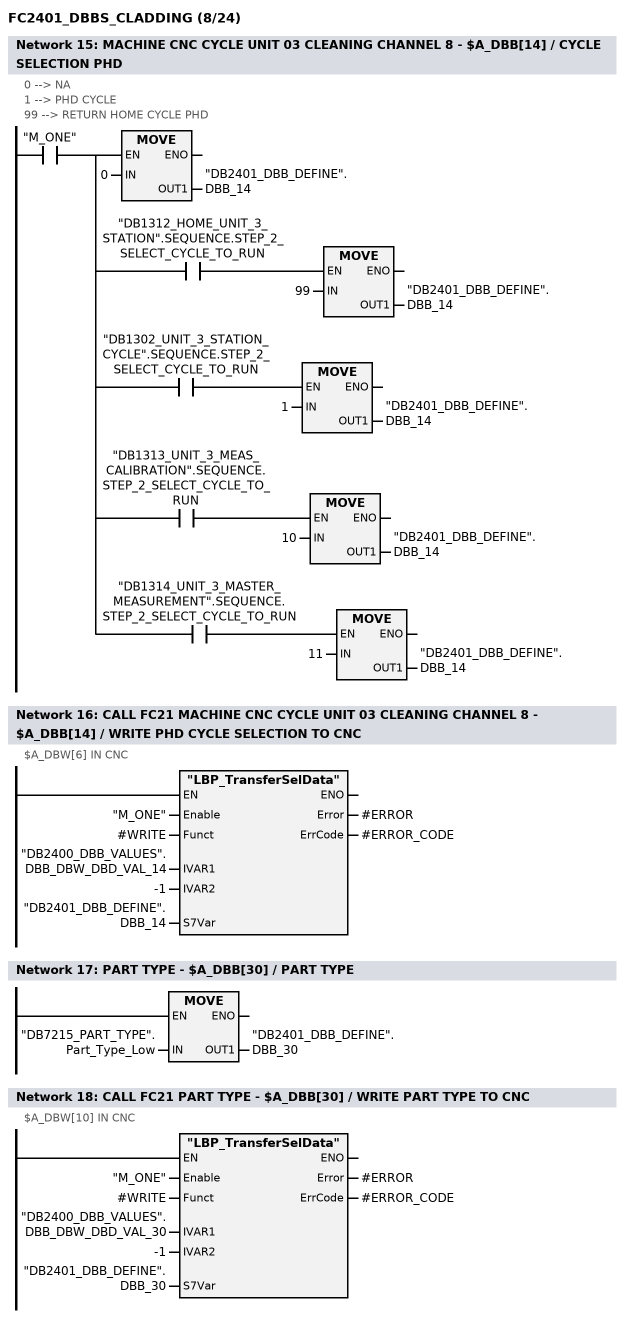
   RUNG wire#powerrail
      Contact( "M_ONE" )
      wire#w1
      { S7_GenerateENO := "TRUE" } Move(in := 0, out1 => "DB2401_DBB_DEFINE".DBB_14)
   END_RUNG
   RUNG wire#w1
      Contact( "DB1312_HOME_UNIT_3_STATION".SEQUENCE.STEP_2_SELECT_CYCLE_TO_RUN )
      { S7_GenerateENO := "TRUE" } Move(in := 99, out1 => "DB2401_DBB_DEFINE".DBB_14)
   END_RUNG
   RUNG wire#w1
      Contact( "DB1302_UNIT_3_STATION_CYCLE".SEQUENCE.STEP_2_SELECT_CYCLE_TO_RUN )
      { S7_GenerateENO := "TRUE" } Move(in := 1, out1 => "DB2401_DBB_DEFINE".DBB_14)
   END_RUNG
   RUNG wire#w1
      Contact( "DB1313_UNIT_3_MEAS_CALIBRATION".SEQUENCE.STEP_2_SELECT_CYCLE_TO_RUN )
      { S7_GenerateENO := "TRUE" } Move(in := 10, out1 => "DB2401_DBB_DEFINE".DBB_14)
   END_RUNG
   RUNG wire#w1
      Contact( "DB1314_UNIT_3_MASTER_MEASUREMENT".SEQUENCE.STEP_2_SELECT_CYCLE_TO_RUN )
      { S7_GenerateENO := "TRUE" } Move(in := 11, out1 => "DB2401_DBB_DEFINE".DBB_14)
   END_RUNG
   // the same network as SCL:
   IF "M_ONE" THEN "DB2401_DBB_DEFINE".DBB_14 := 0; END_IF;
   IF "M_ONE" AND "DB1312_HOME_UNIT_3_STATION".SEQUENCE.STEP_2_SELECT_CYCLE_TO_RUN THEN
       "DB2401_DBB_DEFINE".DBB_14 := 99;
   END_IF;
   IF "M_ONE" AND "DB1302_UNIT_3_STATION_CYCLE".SEQUENCE.STEP_2_SELECT_CYCLE_TO_RUN THEN
       "DB2401_DBB_DEFINE".DBB_14 := 1;
   END_IF;
   IF "M_ONE" AND "DB1313_UNIT_3_MEAS_CALIBRATION".SEQUENCE.STEP_2_SELECT_CYCLE_TO_RUN THEN
       "DB2401_DBB_DEFINE".DBB_14 := 10;
   END_IF;
   IF "M_ONE" AND "DB1314_UNIT_3_MASTER_MEASUREMENT".SEQUENCE.STEP_2_SELECT_CYCLE_TO_RUN THEN
       "DB2401_DBB_DEFINE".DBB_14 := 11;
   END_IF;
END_REGION

REGION Network 16: CALL FC21 MACHINE CNC CYCLE UNIT 03 CLEANING CHANNEL 8 - $A_DBB[14] / WRITE PHD CYCLE SELECTION TO CNC
   // $A_DBW[6] IN CNC
   RUNG wire#powerrail
      "LBP_TransferSelData"(Enable := "M_ONE", Funct := #WRITE, IVAR1 := "DB2400_DBB_VALUES".DBB_DBW_DBD_VAL_14, IVAR2 := -1, S7Var := "DB2401_DBB_DEFINE".DBB_14, Error => #ERROR, ErrCode => #ERROR_CODE)
   END_RUNG
   // the same network as SCL:
   "LBP_TransferSelData"(Enable := "M_ONE",
                         Funct := #WRITE,
                         IVAR1 := "DB2400_DBB_VALUES".DBB_DBW_DBD_VAL_14,
                         IVAR2 := -1,
                         S7Var := "DB2401_DBB_DEFINE".DBB_14,
                         Error => #ERROR,
                         ErrCode => #ERROR_CODE);
END_REGION

REGION Network 17: PART TYPE - $A_DBB[30] / PART TYPE
   RUNG wire#powerrail
      { S7_GenerateENO := "TRUE" } Move(in := "DB7215_PART_TYPE".Part_Type_Low, out1 => "DB2401_DBB_DEFINE".DBB_30)
   END_RUNG
   // the same network as SCL:
   "DB2401_DBB_DEFINE".DBB_30 := "DB7215_PART_TYPE".Part_Type_Low;
END_REGION

REGION Network 18: CALL FC21 PART TYPE - $A_DBB[30] / WRITE PART TYPE TO CNC
   // $A_DBW[10] IN CNC
   RUNG wire#powerrail
      "LBP_TransferSelData"(Enable := "M_ONE", Funct := #WRITE, IVAR1 := "DB2400_DBB_VALUES".DBB_DBW_DBD_VAL_30, IVAR2 := -1, S7Var := "DB2401_DBB_DEFINE".DBB_30, Error => #ERROR, ErrCode => #ERROR_CODE)
   END_RUNG
   // the same network as SCL:
   "LBP_TransferSelData"(Enable := "M_ONE",
                         Funct := #WRITE,
                         IVAR1 := "DB2400_DBB_VALUES".DBB_DBW_DBD_VAL_30,
                         IVAR2 := -1,
                         S7Var := "DB2401_DBB_DEFINE".DBB_30,
                         Error => #ERROR,
                         ErrCode => #ERROR_CODE);
END_REGION

REGION Network 19: FIXTURE NUMBER IN UNIT 01 STATION 1 - $A_DBB[20]
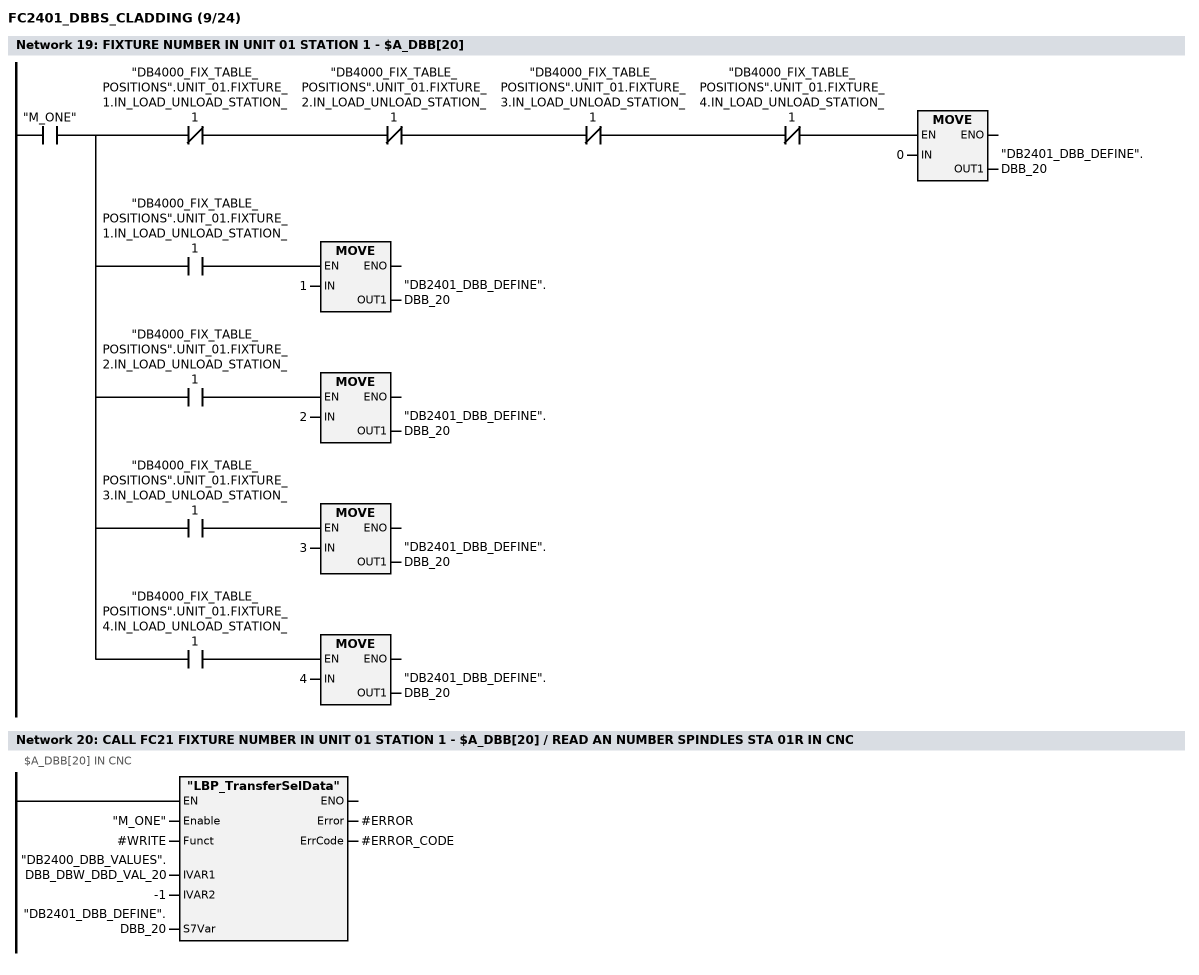
   RUNG wire#powerrail
      Contact( "M_ONE" )
      wire#w1
      I_Contact( "DB4000_FIX_TABLE_POSITIONS".UNIT_01.FIXTURE_1.IN_LOAD_UNLOAD_STATION_1 )
      I_Contact( "DB4000_FIX_TABLE_POSITIONS".UNIT_01.FIXTURE_2.IN_LOAD_UNLOAD_STATION_1 )
      I_Contact( "DB4000_FIX_TABLE_POSITIONS".UNIT_01.FIXTURE_3.IN_LOAD_UNLOAD_STATION_1 )
      I_Contact( "DB4000_FIX_TABLE_POSITIONS".UNIT_01.FIXTURE_4.IN_LOAD_UNLOAD_STATION_1 )
      Move(in := 0, out1 => "DB2401_DBB_DEFINE".DBB_20)
   END_RUNG
   RUNG wire#w1
      Contact( "DB4000_FIX_TABLE_POSITIONS".UNIT_01.FIXTURE_1.IN_LOAD_UNLOAD_STATION_1 )
      Move(in := 1, out1 => "DB2401_DBB_DEFINE".DBB_20)
   END_RUNG
   RUNG wire#w1
      Contact( "DB4000_FIX_TABLE_POSITIONS".UNIT_01.FIXTURE_2.IN_LOAD_UNLOAD_STATION_1 )
      Move(in := 2, out1 => "DB2401_DBB_DEFINE".DBB_20)
   END_RUNG
   RUNG wire#w1
      Contact( "DB4000_FIX_TABLE_POSITIONS".UNIT_01.FIXTURE_3.IN_LOAD_UNLOAD_STATION_1 )
      Move(in := 3, out1 => "DB2401_DBB_DEFINE".DBB_20)
   END_RUNG
   RUNG wire#w1
      Contact( "DB4000_FIX_TABLE_POSITIONS".UNIT_01.FIXTURE_4.IN_LOAD_UNLOAD_STATION_1 )
      Move(in := 4, out1 => "DB2401_DBB_DEFINE".DBB_20)
   END_RUNG
   // the same network as SCL:
   IF "M_ONE" AND NOT "DB4000_FIX_TABLE_POSITIONS".UNIT_01.FIXTURE_1.IN_LOAD_UNLOAD_STATION_1 AND NOT "DB4000_FIX_TABLE_POSITIONS".UNIT_01.FIXTURE_2.IN_LOAD_UNLOAD_STATION_1 AND NOT "DB4000_FIX_TABLE_POSITIONS".UNIT_01.FIXTURE_3.IN_LOAD_UNLOAD_STATION_1 AND NOT "DB4000_FIX_TABLE_POSITIONS".UNIT_01.FIXTURE_4.IN_LOAD_UNLOAD_STATION_1 THEN
       "DB2401_DBB_DEFINE".DBB_20 := 0;
   END_IF;
   IF "M_ONE" AND "DB4000_FIX_TABLE_POSITIONS".UNIT_01.FIXTURE_1.IN_LOAD_UNLOAD_STATION_1 THEN
       "DB2401_DBB_DEFINE".DBB_20 := 1;
   END_IF;
   IF "M_ONE" AND "DB4000_FIX_TABLE_POSITIONS".UNIT_01.FIXTURE_2.IN_LOAD_UNLOAD_STATION_1 THEN
       "DB2401_DBB_DEFINE".DBB_20 := 2;
   END_IF;
   IF "M_ONE" AND "DB4000_FIX_TABLE_POSITIONS".UNIT_01.FIXTURE_3.IN_LOAD_UNLOAD_STATION_1 THEN
       "DB2401_DBB_DEFINE".DBB_20 := 3;
   END_IF;
   IF "M_ONE" AND "DB4000_FIX_TABLE_POSITIONS".UNIT_01.FIXTURE_4.IN_LOAD_UNLOAD_STATION_1 THEN
       "DB2401_DBB_DEFINE".DBB_20 := 4;
   END_IF;
END_REGION

REGION Network 20: CALL FC21 FIXTURE NUMBER IN UNIT 01 STATION 1 - $A_DBB[20] / READ AN NUMBER SPINDLES STA 01R IN CNC
   // $A_DBB[20] IN CNC
   RUNG wire#powerrail
      "LBP_TransferSelData"(Enable := "M_ONE", Funct := #WRITE, IVAR1 := "DB2400_DBB_VALUES".DBB_DBW_DBD_VAL_20, IVAR2 := -1, S7Var := "DB2401_DBB_DEFINE".DBB_20, Error => #ERROR, ErrCode => #ERROR_CODE)
   END_RUNG
   // the same network as SCL:
   "LBP_TransferSelData"(Enable := "M_ONE",
                         Funct := #WRITE,
                         IVAR1 := "DB2400_DBB_VALUES".DBB_DBW_DBD_VAL_20,
                         IVAR2 := -1,
                         S7Var := "DB2401_DBB_DEFINE".DBB_20,
                         Error => #ERROR,
                         ErrCode => #ERROR_CODE);
END_REGION

REGION Network 21: FIXTURE NUMBER IN UNIT 02 STATION 1 - $A_DBB[22]
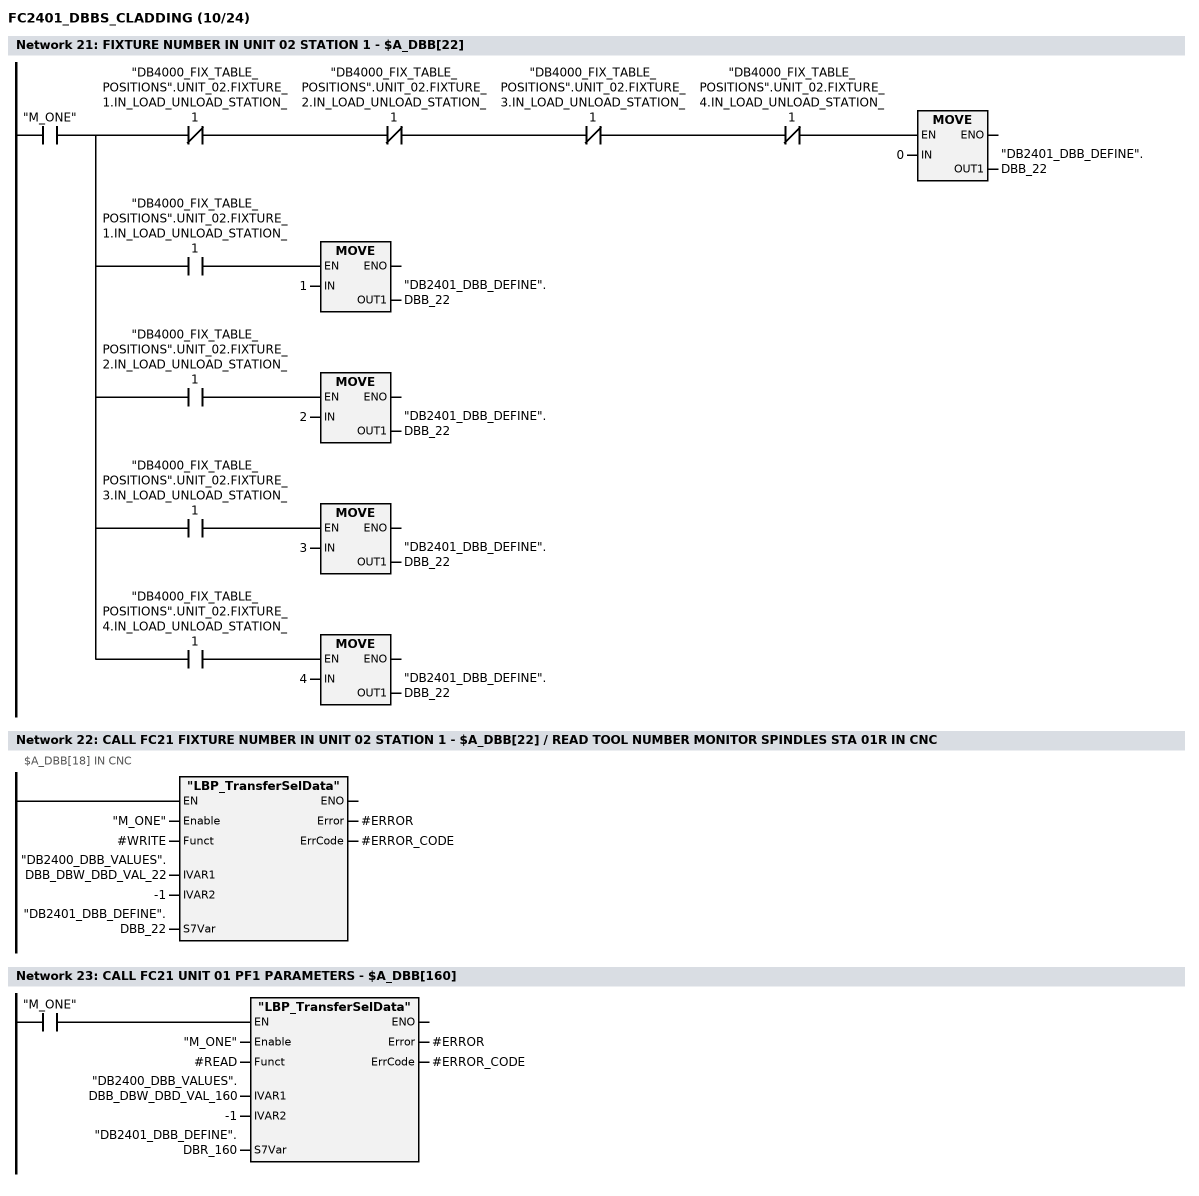
   RUNG wire#powerrail
      Contact( "M_ONE" )
      wire#w1
      I_Contact( "DB4000_FIX_TABLE_POSITIONS".UNIT_02.FIXTURE_1.IN_LOAD_UNLOAD_STATION_1 )
      I_Contact( "DB4000_FIX_TABLE_POSITIONS".UNIT_02.FIXTURE_2.IN_LOAD_UNLOAD_STATION_1 )
      I_Contact( "DB4000_FIX_TABLE_POSITIONS".UNIT_02.FIXTURE_3.IN_LOAD_UNLOAD_STATION_1 )
      I_Contact( "DB4000_FIX_TABLE_POSITIONS".UNIT_02.FIXTURE_4.IN_LOAD_UNLOAD_STATION_1 )
      Move(in := 0, out1 => "DB2401_DBB_DEFINE".DBB_22)
   END_RUNG
   RUNG wire#w1
      Contact( "DB4000_FIX_TABLE_POSITIONS".UNIT_02.FIXTURE_1.IN_LOAD_UNLOAD_STATION_1 )
      Move(in := 1, out1 => "DB2401_DBB_DEFINE".DBB_22)
   END_RUNG
   RUNG wire#w1
      Contact( "DB4000_FIX_TABLE_POSITIONS".UNIT_02.FIXTURE_2.IN_LOAD_UNLOAD_STATION_1 )
      Move(in := 2, out1 => "DB2401_DBB_DEFINE".DBB_22)
   END_RUNG
   RUNG wire#w1
      Contact( "DB4000_FIX_TABLE_POSITIONS".UNIT_02.FIXTURE_3.IN_LOAD_UNLOAD_STATION_1 )
      Move(in := 3, out1 => "DB2401_DBB_DEFINE".DBB_22)
   END_RUNG
   RUNG wire#w1
      Contact( "DB4000_FIX_TABLE_POSITIONS".UNIT_02.FIXTURE_4.IN_LOAD_UNLOAD_STATION_1 )
      Move(in := 4, out1 => "DB2401_DBB_DEFINE".DBB_22)
   END_RUNG
   // the same network as SCL:
   IF "M_ONE" AND NOT "DB4000_FIX_TABLE_POSITIONS".UNIT_02.FIXTURE_1.IN_LOAD_UNLOAD_STATION_1 AND NOT "DB4000_FIX_TABLE_POSITIONS".UNIT_02.FIXTURE_2.IN_LOAD_UNLOAD_STATION_1 AND NOT "DB4000_FIX_TABLE_POSITIONS".UNIT_02.FIXTURE_3.IN_LOAD_UNLOAD_STATION_1 AND NOT "DB4000_FIX_TABLE_POSITIONS".UNIT_02.FIXTURE_4.IN_LOAD_UNLOAD_STATION_1 THEN
       "DB2401_DBB_DEFINE".DBB_22 := 0;
   END_IF;
   IF "M_ONE" AND "DB4000_FIX_TABLE_POSITIONS".UNIT_02.FIXTURE_1.IN_LOAD_UNLOAD_STATION_1 THEN
       "DB2401_DBB_DEFINE".DBB_22 := 1;
   END_IF;
   IF "M_ONE" AND "DB4000_FIX_TABLE_POSITIONS".UNIT_02.FIXTURE_2.IN_LOAD_UNLOAD_STATION_1 THEN
       "DB2401_DBB_DEFINE".DBB_22 := 2;
   END_IF;
   IF "M_ONE" AND "DB4000_FIX_TABLE_POSITIONS".UNIT_02.FIXTURE_3.IN_LOAD_UNLOAD_STATION_1 THEN
       "DB2401_DBB_DEFINE".DBB_22 := 3;
   END_IF;
   IF "M_ONE" AND "DB4000_FIX_TABLE_POSITIONS".UNIT_02.FIXTURE_4.IN_LOAD_UNLOAD_STATION_1 THEN
       "DB2401_DBB_DEFINE".DBB_22 := 4;
   END_IF;
END_REGION

REGION Network 22: CALL FC21 FIXTURE NUMBER IN UNIT 02 STATION 1 - $A_DBB[22] / READ TOOL NUMBER MONITOR SPINDLES STA 01R IN CNC
   // $A_DBB[18] IN CNC
   RUNG wire#powerrail
      "LBP_TransferSelData"(Enable := "M_ONE", Funct := #WRITE, IVAR1 := "DB2400_DBB_VALUES".DBB_DBW_DBD_VAL_22, IVAR2 := -1, S7Var := "DB2401_DBB_DEFINE".DBB_22, Error => #ERROR, ErrCode => #ERROR_CODE)
   END_RUNG
   // the same network as SCL:
   "LBP_TransferSelData"(Enable := "M_ONE",
                         Funct := #WRITE,
                         IVAR1 := "DB2400_DBB_VALUES".DBB_DBW_DBD_VAL_22,
                         IVAR2 := -1,
                         S7Var := "DB2401_DBB_DEFINE".DBB_22,
                         Error => #ERROR,
                         ErrCode => #ERROR_CODE);
END_REGION

REGION Network 23: CALL FC21 UNIT 01 PF1 PARAMETERS - $A_DBB[160]
   RUNG wire#powerrail
      Contact( "M_ONE" )
      "LBP_TransferSelData"(Enable := "M_ONE", Funct := #READ, IVAR1 := "DB2400_DBB_VALUES".DBB_DBW_DBD_VAL_160, IVAR2 := -1, S7Var := "DB2401_DBB_DEFINE".DBR_160, Error => #ERROR, ErrCode => #ERROR_CODE)
   END_RUNG
   // the same network as SCL:
   IF "M_ONE" THEN
       "LBP_TransferSelData"(Enable := "M_ONE",
                             Funct := #READ,
                             IVAR1 := "DB2400_DBB_VALUES".DBB_DBW_DBD_VAL_160,
                             IVAR2 := -1,
                             S7Var := "DB2401_DBB_DEFINE".DBR_160,
                             Error => #ERROR,
                             ErrCode => #ERROR_CODE);
   END_IF;
END_REGION

REGION Network 24: CALL FC21 UNIT 01 PF1 PARAMETERS - $A_DBB[164]
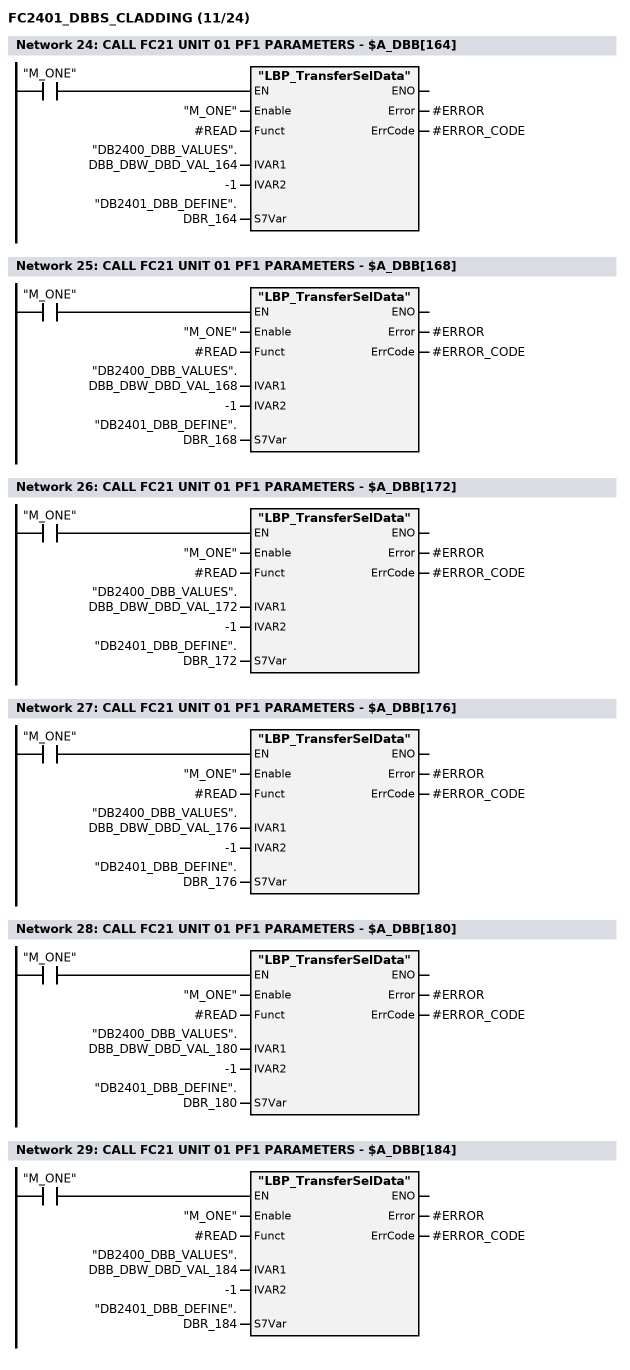
   RUNG wire#powerrail
      Contact( "M_ONE" )
      "LBP_TransferSelData"(Enable := "M_ONE", Funct := #READ, IVAR1 := "DB2400_DBB_VALUES".DBB_DBW_DBD_VAL_164, IVAR2 := -1, S7Var := "DB2401_DBB_DEFINE".DBR_164, Error => #ERROR, ErrCode => #ERROR_CODE)
   END_RUNG
   // the same network as SCL:
   IF "M_ONE" THEN
       "LBP_TransferSelData"(Enable := "M_ONE",
                             Funct := #READ,
                             IVAR1 := "DB2400_DBB_VALUES".DBB_DBW_DBD_VAL_164,
                             IVAR2 := -1,
                             S7Var := "DB2401_DBB_DEFINE".DBR_164,
                             Error => #ERROR,
                             ErrCode => #ERROR_CODE);
   END_IF;
END_REGION

REGION Network 25: CALL FC21 UNIT 01 PF1 PARAMETERS - $A_DBB[168]
   RUNG wire#powerrail
      Contact( "M_ONE" )
      "LBP_TransferSelData"(Enable := "M_ONE", Funct := #READ, IVAR1 := "DB2400_DBB_VALUES".DBB_DBW_DBD_VAL_168, IVAR2 := -1, S7Var := "DB2401_DBB_DEFINE".DBR_168, Error => #ERROR, ErrCode => #ERROR_CODE)
   END_RUNG
   // the same network as SCL:
   IF "M_ONE" THEN
       "LBP_TransferSelData"(Enable := "M_ONE",
                             Funct := #READ,
                             IVAR1 := "DB2400_DBB_VALUES".DBB_DBW_DBD_VAL_168,
                             IVAR2 := -1,
                             S7Var := "DB2401_DBB_DEFINE".DBR_168,
                             Error => #ERROR,
                             ErrCode => #ERROR_CODE);
   END_IF;
END_REGION

REGION Network 26: CALL FC21 UNIT 01 PF1 PARAMETERS - $A_DBB[172]
   RUNG wire#powerrail
      Contact( "M_ONE" )
      "LBP_TransferSelData"(Enable := "M_ONE", Funct := #READ, IVAR1 := "DB2400_DBB_VALUES".DBB_DBW_DBD_VAL_172, IVAR2 := -1, S7Var := "DB2401_DBB_DEFINE".DBR_172, Error => #ERROR, ErrCode => #ERROR_CODE)
   END_RUNG
   // the same network as SCL:
   IF "M_ONE" THEN
       "LBP_TransferSelData"(Enable := "M_ONE",
                             Funct := #READ,
                             IVAR1 := "DB2400_DBB_VALUES".DBB_DBW_DBD_VAL_172,
                             IVAR2 := -1,
                             S7Var := "DB2401_DBB_DEFINE".DBR_172,
                             Error => #ERROR,
                             ErrCode => #ERROR_CODE);
   END_IF;
END_REGION

REGION Network 27: CALL FC21 UNIT 01 PF1 PARAMETERS - $A_DBB[176]
   RUNG wire#powerrail
      Contact( "M_ONE" )
      "LBP_TransferSelData"(Enable := "M_ONE", Funct := #READ, IVAR1 := "DB2400_DBB_VALUES".DBB_DBW_DBD_VAL_176, IVAR2 := -1, S7Var := "DB2401_DBB_DEFINE".DBR_176, Error => #ERROR, ErrCode => #ERROR_CODE)
   END_RUNG
   // the same network as SCL:
   IF "M_ONE" THEN
       "LBP_TransferSelData"(Enable := "M_ONE",
                             Funct := #READ,
                             IVAR1 := "DB2400_DBB_VALUES".DBB_DBW_DBD_VAL_176,
                             IVAR2 := -1,
                             S7Var := "DB2401_DBB_DEFINE".DBR_176,
                             Error => #ERROR,
                             ErrCode => #ERROR_CODE);
   END_IF;
END_REGION

REGION Network 28: CALL FC21 UNIT 01 PF1 PARAMETERS - $A_DBB[180]
   RUNG wire#powerrail
      Contact( "M_ONE" )
      "LBP_TransferSelData"(Enable := "M_ONE", Funct := #READ, IVAR1 := "DB2400_DBB_VALUES".DBB_DBW_DBD_VAL_180, IVAR2 := -1, S7Var := "DB2401_DBB_DEFINE".DBR_180, Error => #ERROR, ErrCode => #ERROR_CODE)
   END_RUNG
   // the same network as SCL:
   IF "M_ONE" THEN
       "LBP_TransferSelData"(Enable := "M_ONE",
                             Funct := #READ,
                             IVAR1 := "DB2400_DBB_VALUES".DBB_DBW_DBD_VAL_180,
                             IVAR2 := -1,
                             S7Var := "DB2401_DBB_DEFINE".DBR_180,
                             Error => #ERROR,
                             ErrCode => #ERROR_CODE);
   END_IF;
END_REGION

REGION Network 29: CALL FC21 UNIT 01 PF1 PARAMETERS - $A_DBB[184]
   RUNG wire#powerrail
      Contact( "M_ONE" )
      "LBP_TransferSelData"(Enable := "M_ONE", Funct := #READ, IVAR1 := "DB2400_DBB_VALUES".DBB_DBW_DBD_VAL_184, IVAR2 := -1, S7Var := "DB2401_DBB_DEFINE".DBR_184, Error => #ERROR, ErrCode => #ERROR_CODE)
   END_RUNG
   // the same network as SCL:
   IF "M_ONE" THEN
       "LBP_TransferSelData"(Enable := "M_ONE",
                             Funct := #READ,
                             IVAR1 := "DB2400_DBB_VALUES".DBB_DBW_DBD_VAL_184,
                             IVAR2 := -1,
                             S7Var := "DB2401_DBB_DEFINE".DBR_184,
                             Error => #ERROR,
                             ErrCode => #ERROR_CODE);
   END_IF;
END_REGION

REGION Network 30: CALL FC21 UNIT 01 PF1 PARAMETERS - $A_DBB[188]
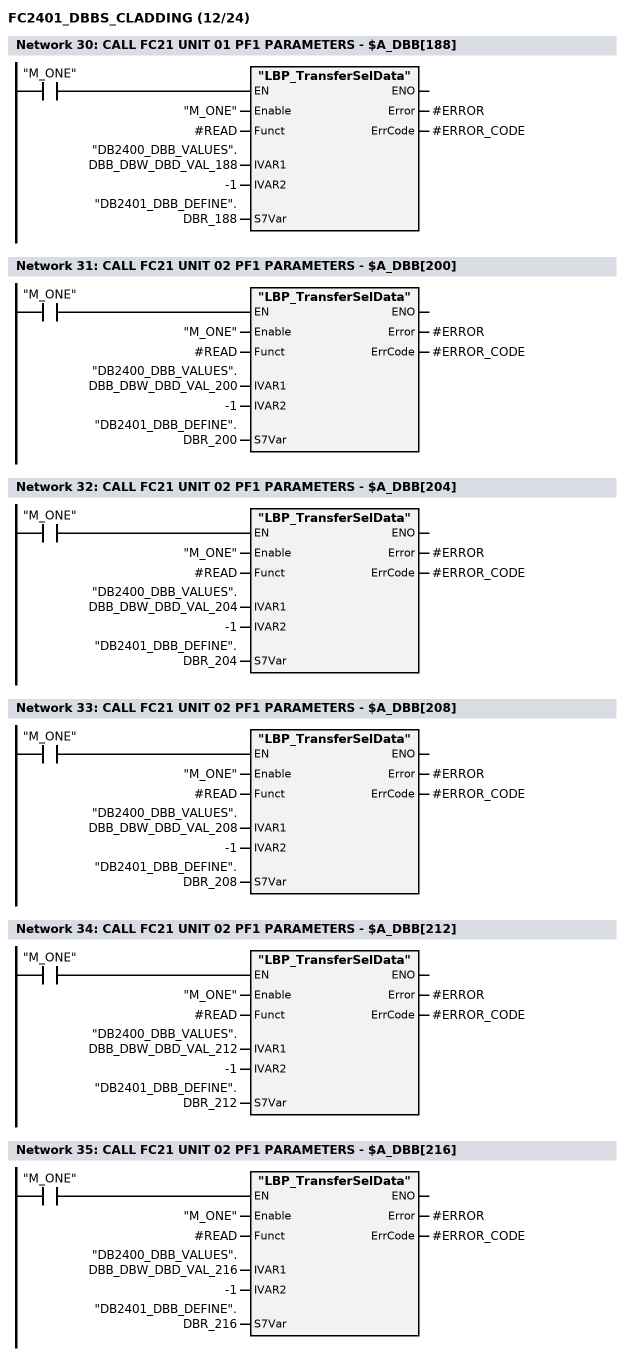
   RUNG wire#powerrail
      Contact( "M_ONE" )
      "LBP_TransferSelData"(Enable := "M_ONE", Funct := #READ, IVAR1 := "DB2400_DBB_VALUES".DBB_DBW_DBD_VAL_188, IVAR2 := -1, S7Var := "DB2401_DBB_DEFINE".DBR_188, Error => #ERROR, ErrCode => #ERROR_CODE)
   END_RUNG
   // the same network as SCL:
   IF "M_ONE" THEN
       "LBP_TransferSelData"(Enable := "M_ONE",
                             Funct := #READ,
                             IVAR1 := "DB2400_DBB_VALUES".DBB_DBW_DBD_VAL_188,
                             IVAR2 := -1,
                             S7Var := "DB2401_DBB_DEFINE".DBR_188,
                             Error => #ERROR,
                             ErrCode => #ERROR_CODE);
   END_IF;
END_REGION

REGION Network 31: CALL FC21 UNIT 02 PF1 PARAMETERS - $A_DBB[200]
   RUNG wire#powerrail
      Contact( "M_ONE" )
      "LBP_TransferSelData"(Enable := "M_ONE", Funct := #READ, IVAR1 := "DB2400_DBB_VALUES".DBB_DBW_DBD_VAL_200, IVAR2 := -1, S7Var := "DB2401_DBB_DEFINE".DBR_200, Error => #ERROR, ErrCode => #ERROR_CODE)
   END_RUNG
   // the same network as SCL:
   IF "M_ONE" THEN
       "LBP_TransferSelData"(Enable := "M_ONE",
                             Funct := #READ,
                             IVAR1 := "DB2400_DBB_VALUES".DBB_DBW_DBD_VAL_200,
                             IVAR2 := -1,
                             S7Var := "DB2401_DBB_DEFINE".DBR_200,
                             Error => #ERROR,
                             ErrCode => #ERROR_CODE);
   END_IF;
END_REGION

REGION Network 32: CALL FC21 UNIT 02 PF1 PARAMETERS - $A_DBB[204]
   RUNG wire#powerrail
      Contact( "M_ONE" )
      "LBP_TransferSelData"(Enable := "M_ONE", Funct := #READ, IVAR1 := "DB2400_DBB_VALUES".DBB_DBW_DBD_VAL_204, IVAR2 := -1, S7Var := "DB2401_DBB_DEFINE".DBR_204, Error => #ERROR, ErrCode => #ERROR_CODE)
   END_RUNG
   // the same network as SCL:
   IF "M_ONE" THEN
       "LBP_TransferSelData"(Enable := "M_ONE",
                             Funct := #READ,
                             IVAR1 := "DB2400_DBB_VALUES".DBB_DBW_DBD_VAL_204,
                             IVAR2 := -1,
                             S7Var := "DB2401_DBB_DEFINE".DBR_204,
                             Error => #ERROR,
                             ErrCode => #ERROR_CODE);
   END_IF;
END_REGION

REGION Network 33: CALL FC21 UNIT 02 PF1 PARAMETERS - $A_DBB[208]
   RUNG wire#powerrail
      Contact( "M_ONE" )
      "LBP_TransferSelData"(Enable := "M_ONE", Funct := #READ, IVAR1 := "DB2400_DBB_VALUES".DBB_DBW_DBD_VAL_208, IVAR2 := -1, S7Var := "DB2401_DBB_DEFINE".DBR_208, Error => #ERROR, ErrCode => #ERROR_CODE)
   END_RUNG
   // the same network as SCL:
   IF "M_ONE" THEN
       "LBP_TransferSelData"(Enable := "M_ONE",
                             Funct := #READ,
                             IVAR1 := "DB2400_DBB_VALUES".DBB_DBW_DBD_VAL_208,
                             IVAR2 := -1,
                             S7Var := "DB2401_DBB_DEFINE".DBR_208,
                             Error => #ERROR,
                             ErrCode => #ERROR_CODE);
   END_IF;
END_REGION

REGION Network 34: CALL FC21 UNIT 02 PF1 PARAMETERS - $A_DBB[212]
   RUNG wire#powerrail
      Contact( "M_ONE" )
      "LBP_TransferSelData"(Enable := "M_ONE", Funct := #READ, IVAR1 := "DB2400_DBB_VALUES".DBB_DBW_DBD_VAL_212, IVAR2 := -1, S7Var := "DB2401_DBB_DEFINE".DBR_212, Error => #ERROR, ErrCode => #ERROR_CODE)
   END_RUNG
   // the same network as SCL:
   IF "M_ONE" THEN
       "LBP_TransferSelData"(Enable := "M_ONE",
                             Funct := #READ,
                             IVAR1 := "DB2400_DBB_VALUES".DBB_DBW_DBD_VAL_212,
                             IVAR2 := -1,
                             S7Var := "DB2401_DBB_DEFINE".DBR_212,
                             Error => #ERROR,
                             ErrCode => #ERROR_CODE);
   END_IF;
END_REGION

REGION Network 35: CALL FC21 UNIT 02 PF1 PARAMETERS - $A_DBB[216]
   RUNG wire#powerrail
      Contact( "M_ONE" )
      "LBP_TransferSelData"(Enable := "M_ONE", Funct := #READ, IVAR1 := "DB2400_DBB_VALUES".DBB_DBW_DBD_VAL_216, IVAR2 := -1, S7Var := "DB2401_DBB_DEFINE".DBR_216, Error => #ERROR, ErrCode => #ERROR_CODE)
   END_RUNG
   // the same network as SCL:
   IF "M_ONE" THEN
       "LBP_TransferSelData"(Enable := "M_ONE",
                             Funct := #READ,
                             IVAR1 := "DB2400_DBB_VALUES".DBB_DBW_DBD_VAL_216,
                             IVAR2 := -1,
                             S7Var := "DB2401_DBB_DEFINE".DBR_216,
                             Error => #ERROR,
                             ErrCode => #ERROR_CODE);
   END_IF;
END_REGION

REGION Network 36: CALL FC21 UNIT 02 PF1 PARAMETERS - $A_DBB[220]
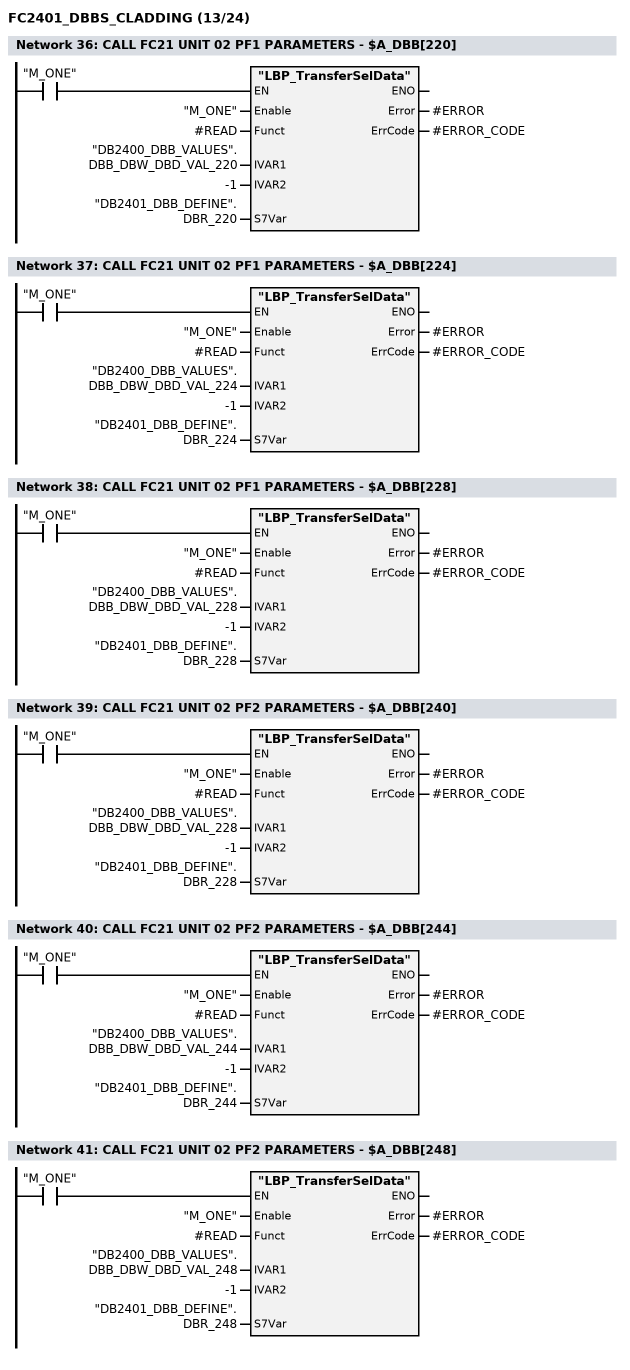
   RUNG wire#powerrail
      Contact( "M_ONE" )
      "LBP_TransferSelData"(Enable := "M_ONE", Funct := #READ, IVAR1 := "DB2400_DBB_VALUES".DBB_DBW_DBD_VAL_220, IVAR2 := -1, S7Var := "DB2401_DBB_DEFINE".DBR_220, Error => #ERROR, ErrCode => #ERROR_CODE)
   END_RUNG
   // the same network as SCL:
   IF "M_ONE" THEN
       "LBP_TransferSelData"(Enable := "M_ONE",
                             Funct := #READ,
                             IVAR1 := "DB2400_DBB_VALUES".DBB_DBW_DBD_VAL_220,
                             IVAR2 := -1,
                             S7Var := "DB2401_DBB_DEFINE".DBR_220,
                             Error => #ERROR,
                             ErrCode => #ERROR_CODE);
   END_IF;
END_REGION

REGION Network 37: CALL FC21 UNIT 02 PF1 PARAMETERS - $A_DBB[224]
   RUNG wire#powerrail
      Contact( "M_ONE" )
      "LBP_TransferSelData"(Enable := "M_ONE", Funct := #READ, IVAR1 := "DB2400_DBB_VALUES".DBB_DBW_DBD_VAL_224, IVAR2 := -1, S7Var := "DB2401_DBB_DEFINE".DBR_224, Error => #ERROR, ErrCode => #ERROR_CODE)
   END_RUNG
   // the same network as SCL:
   IF "M_ONE" THEN
       "LBP_TransferSelData"(Enable := "M_ONE",
                             Funct := #READ,
                             IVAR1 := "DB2400_DBB_VALUES".DBB_DBW_DBD_VAL_224,
                             IVAR2 := -1,
                             S7Var := "DB2401_DBB_DEFINE".DBR_224,
                             Error => #ERROR,
                             ErrCode => #ERROR_CODE);
   END_IF;
END_REGION

REGION Network 38: CALL FC21 UNIT 02 PF1 PARAMETERS - $A_DBB[228]
   RUNG wire#powerrail
      Contact( "M_ONE" )
      "LBP_TransferSelData"(Enable := "M_ONE", Funct := #READ, IVAR1 := "DB2400_DBB_VALUES".DBB_DBW_DBD_VAL_228, IVAR2 := -1, S7Var := "DB2401_DBB_DEFINE".DBR_228, Error => #ERROR, ErrCode => #ERROR_CODE)
   END_RUNG
   // the same network as SCL:
   IF "M_ONE" THEN
       "LBP_TransferSelData"(Enable := "M_ONE",
                             Funct := #READ,
                             IVAR1 := "DB2400_DBB_VALUES".DBB_DBW_DBD_VAL_228,
                             IVAR2 := -1,
                             S7Var := "DB2401_DBB_DEFINE".DBR_228,
                             Error => #ERROR,
                             ErrCode => #ERROR_CODE);
   END_IF;
END_REGION

REGION Network 39: CALL FC21 UNIT 02 PF2 PARAMETERS - $A_DBB[240]
   RUNG wire#powerrail
      Contact( "M_ONE" )
      "LBP_TransferSelData"(Enable := "M_ONE", Funct := #READ, IVAR1 := "DB2400_DBB_VALUES".DBB_DBW_DBD_VAL_228, IVAR2 := -1, S7Var := "DB2401_DBB_DEFINE".DBR_228, Error => #ERROR, ErrCode => #ERROR_CODE)
   END_RUNG
   // the same network as SCL:
   IF "M_ONE" THEN
       "LBP_TransferSelData"(Enable := "M_ONE",
                             Funct := #READ,
                             IVAR1 := "DB2400_DBB_VALUES".DBB_DBW_DBD_VAL_228,
                             IVAR2 := -1,
                             S7Var := "DB2401_DBB_DEFINE".DBR_228,
                             Error => #ERROR,
                             ErrCode => #ERROR_CODE);
   END_IF;
END_REGION

REGION Network 40: CALL FC21 UNIT 02 PF2 PARAMETERS - $A_DBB[244]
   RUNG wire#powerrail
      Contact( "M_ONE" )
      "LBP_TransferSelData"(Enable := "M_ONE", Funct := #READ, IVAR1 := "DB2400_DBB_VALUES".DBB_DBW_DBD_VAL_244, IVAR2 := -1, S7Var := "DB2401_DBB_DEFINE".DBR_244, Error => #ERROR, ErrCode => #ERROR_CODE)
   END_RUNG
   // the same network as SCL:
   IF "M_ONE" THEN
       "LBP_TransferSelData"(Enable := "M_ONE",
                             Funct := #READ,
                             IVAR1 := "DB2400_DBB_VALUES".DBB_DBW_DBD_VAL_244,
                             IVAR2 := -1,
                             S7Var := "DB2401_DBB_DEFINE".DBR_244,
                             Error => #ERROR,
                             ErrCode => #ERROR_CODE);
   END_IF;
END_REGION

REGION Network 41: CALL FC21 UNIT 02 PF2 PARAMETERS - $A_DBB[248]
   RUNG wire#powerrail
      Contact( "M_ONE" )
      "LBP_TransferSelData"(Enable := "M_ONE", Funct := #READ, IVAR1 := "DB2400_DBB_VALUES".DBB_DBW_DBD_VAL_248, IVAR2 := -1, S7Var := "DB2401_DBB_DEFINE".DBR_248, Error => #ERROR, ErrCode => #ERROR_CODE)
   END_RUNG
   // the same network as SCL:
   IF "M_ONE" THEN
       "LBP_TransferSelData"(Enable := "M_ONE",
                             Funct := #READ,
                             IVAR1 := "DB2400_DBB_VALUES".DBB_DBW_DBD_VAL_248,
                             IVAR2 := -1,
                             S7Var := "DB2401_DBB_DEFINE".DBR_248,
                             Error => #ERROR,
                             ErrCode => #ERROR_CODE);
   END_IF;
END_REGION

REGION Network 42: CALL FC21 UNIT 02 PF2 PARAMETERS - $A_DBB[252]
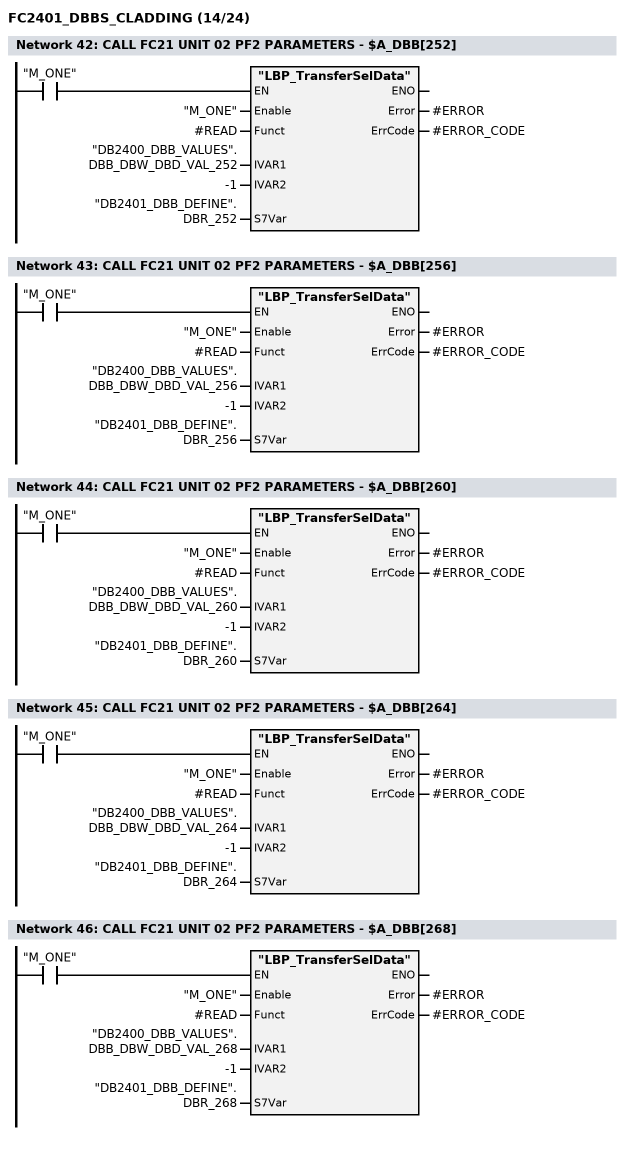
   RUNG wire#powerrail
      Contact( "M_ONE" )
      "LBP_TransferSelData"(Enable := "M_ONE", Funct := #READ, IVAR1 := "DB2400_DBB_VALUES".DBB_DBW_DBD_VAL_252, IVAR2 := -1, S7Var := "DB2401_DBB_DEFINE".DBR_252, Error => #ERROR, ErrCode => #ERROR_CODE)
   END_RUNG
   // the same network as SCL:
   IF "M_ONE" THEN
       "LBP_TransferSelData"(Enable := "M_ONE",
                             Funct := #READ,
                             IVAR1 := "DB2400_DBB_VALUES".DBB_DBW_DBD_VAL_252,
                             IVAR2 := -1,
                             S7Var := "DB2401_DBB_DEFINE".DBR_252,
                             Error => #ERROR,
                             ErrCode => #ERROR_CODE);
   END_IF;
END_REGION

REGION Network 43: CALL FC21 UNIT 02 PF2 PARAMETERS - $A_DBB[256]
   RUNG wire#powerrail
      Contact( "M_ONE" )
      "LBP_TransferSelData"(Enable := "M_ONE", Funct := #READ, IVAR1 := "DB2400_DBB_VALUES".DBB_DBW_DBD_VAL_256, IVAR2 := -1, S7Var := "DB2401_DBB_DEFINE".DBR_256, Error => #ERROR, ErrCode => #ERROR_CODE)
   END_RUNG
   // the same network as SCL:
   IF "M_ONE" THEN
       "LBP_TransferSelData"(Enable := "M_ONE",
                             Funct := #READ,
                             IVAR1 := "DB2400_DBB_VALUES".DBB_DBW_DBD_VAL_256,
                             IVAR2 := -1,
                             S7Var := "DB2401_DBB_DEFINE".DBR_256,
                             Error => #ERROR,
                             ErrCode => #ERROR_CODE);
   END_IF;
END_REGION

REGION Network 44: CALL FC21 UNIT 02 PF2 PARAMETERS - $A_DBB[260]
   RUNG wire#powerrail
      Contact( "M_ONE" )
      "LBP_TransferSelData"(Enable := "M_ONE", Funct := #READ, IVAR1 := "DB2400_DBB_VALUES".DBB_DBW_DBD_VAL_260, IVAR2 := -1, S7Var := "DB2401_DBB_DEFINE".DBR_260, Error => #ERROR, ErrCode => #ERROR_CODE)
   END_RUNG
   // the same network as SCL:
   IF "M_ONE" THEN
       "LBP_TransferSelData"(Enable := "M_ONE",
                             Funct := #READ,
                             IVAR1 := "DB2400_DBB_VALUES".DBB_DBW_DBD_VAL_260,
                             IVAR2 := -1,
                             S7Var := "DB2401_DBB_DEFINE".DBR_260,
                             Error => #ERROR,
                             ErrCode => #ERROR_CODE);
   END_IF;
END_REGION

REGION Network 45: CALL FC21 UNIT 02 PF2 PARAMETERS - $A_DBB[264]
   RUNG wire#powerrail
      Contact( "M_ONE" )
      "LBP_TransferSelData"(Enable := "M_ONE", Funct := #READ, IVAR1 := "DB2400_DBB_VALUES".DBB_DBW_DBD_VAL_264, IVAR2 := -1, S7Var := "DB2401_DBB_DEFINE".DBR_264, Error => #ERROR, ErrCode => #ERROR_CODE)
   END_RUNG
   // the same network as SCL:
   IF "M_ONE" THEN
       "LBP_TransferSelData"(Enable := "M_ONE",
                             Funct := #READ,
                             IVAR1 := "DB2400_DBB_VALUES".DBB_DBW_DBD_VAL_264,
                             IVAR2 := -1,
                             S7Var := "DB2401_DBB_DEFINE".DBR_264,
                             Error => #ERROR,
                             ErrCode => #ERROR_CODE);
   END_IF;
END_REGION

REGION Network 46: CALL FC21 UNIT 02 PF2 PARAMETERS - $A_DBB[268]
   RUNG wire#powerrail
      Contact( "M_ONE" )
      "LBP_TransferSelData"(Enable := "M_ONE", Funct := #READ, IVAR1 := "DB2400_DBB_VALUES".DBB_DBW_DBD_VAL_268, IVAR2 := -1, S7Var := "DB2401_DBB_DEFINE".DBR_268, Error => #ERROR, ErrCode => #ERROR_CODE)
   END_RUNG
   // the same network as SCL:
   IF "M_ONE" THEN
       "LBP_TransferSelData"(Enable := "M_ONE",
                             Funct := #READ,
                             IVAR1 := "DB2400_DBB_VALUES".DBB_DBW_DBD_VAL_268,
                             IVAR2 := -1,
                             S7Var := "DB2401_DBB_DEFINE".DBR_268,
                             Error => #ERROR,
                             ErrCode => #ERROR_CODE);
   END_IF;
END_REGION

REGION Network 47: CALL FC21 UNIT 01 LASER POWER - $A_DBB[504] / READ TOOL NUMBER MONITOR SPINDLES STA 01R IN CNC
   // $A_DBB[18] IN CNC
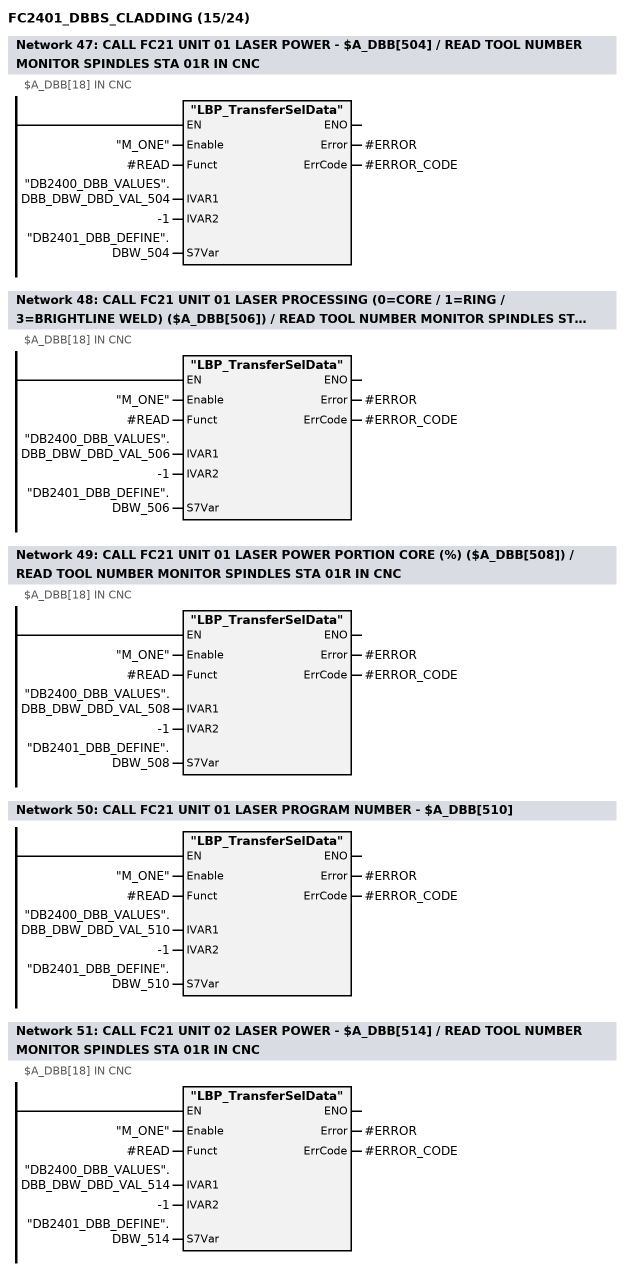
   RUNG wire#powerrail
      "LBP_TransferSelData"(Enable := "M_ONE", Funct := #READ, IVAR1 := "DB2400_DBB_VALUES".DBB_DBW_DBD_VAL_504, IVAR2 := -1, S7Var := "DB2401_DBB_DEFINE".DBW_504, Error => #ERROR, ErrCode => #ERROR_CODE)
   END_RUNG
   // the same network as SCL:
   "LBP_TransferSelData"(Enable := "M_ONE",
                         Funct := #READ,
                         IVAR1 := "DB2400_DBB_VALUES".DBB_DBW_DBD_VAL_504,
                         IVAR2 := -1,
                         S7Var := "DB2401_DBB_DEFINE".DBW_504,
                         Error => #ERROR,
                         ErrCode => #ERROR_CODE);
END_REGION

REGION Network 48: CALL FC21 UNIT 01 LASER PROCESSING (0=CORE / 1=RING / 3=BRIGHTLINE WELD) ($A_DBB[506]) / READ TOOL NUMBER MONITOR SPINDLES STA 01R IN CNC
   // $A_DBB[18] IN CNC
   RUNG wire#powerrail
      "LBP_TransferSelData"(Enable := "M_ONE", Funct := #READ, IVAR1 := "DB2400_DBB_VALUES".DBB_DBW_DBD_VAL_506, IVAR2 := -1, S7Var := "DB2401_DBB_DEFINE".DBW_506, Error => #ERROR, ErrCode => #ERROR_CODE)
   END_RUNG
   // the same network as SCL:
   "LBP_TransferSelData"(Enable := "M_ONE",
                         Funct := #READ,
                         IVAR1 := "DB2400_DBB_VALUES".DBB_DBW_DBD_VAL_506,
                         IVAR2 := -1,
                         S7Var := "DB2401_DBB_DEFINE".DBW_506,
                         Error => #ERROR,
                         ErrCode => #ERROR_CODE);
END_REGION

REGION Network 49: CALL FC21 UNIT 01 LASER POWER PORTION CORE (%) ($A_DBB[508]) / READ TOOL NUMBER MONITOR SPINDLES STA 01R IN CNC
   // $A_DBB[18] IN CNC
   RUNG wire#powerrail
      "LBP_TransferSelData"(Enable := "M_ONE", Funct := #READ, IVAR1 := "DB2400_DBB_VALUES".DBB_DBW_DBD_VAL_508, IVAR2 := -1, S7Var := "DB2401_DBB_DEFINE".DBW_508, Error => #ERROR, ErrCode => #ERROR_CODE)
   END_RUNG
   // the same network as SCL:
   "LBP_TransferSelData"(Enable := "M_ONE",
                         Funct := #READ,
                         IVAR1 := "DB2400_DBB_VALUES".DBB_DBW_DBD_VAL_508,
                         IVAR2 := -1,
                         S7Var := "DB2401_DBB_DEFINE".DBW_508,
                         Error => #ERROR,
                         ErrCode => #ERROR_CODE);
END_REGION

REGION Network 50: CALL FC21 UNIT 01 LASER PROGRAM NUMBER - $A_DBB[510]
   RUNG wire#powerrail
      "LBP_TransferSelData"(Enable := "M_ONE", Funct := #READ, IVAR1 := "DB2400_DBB_VALUES".DBB_DBW_DBD_VAL_510, IVAR2 := -1, S7Var := "DB2401_DBB_DEFINE".DBW_510, Error => #ERROR, ErrCode => #ERROR_CODE)
   END_RUNG
   // the same network as SCL:
   "LBP_TransferSelData"(Enable := "M_ONE",
                         Funct := #READ,
                         IVAR1 := "DB2400_DBB_VALUES".DBB_DBW_DBD_VAL_510,
                         IVAR2 := -1,
                         S7Var := "DB2401_DBB_DEFINE".DBW_510,
                         Error => #ERROR,
                         ErrCode => #ERROR_CODE);
END_REGION

REGION Network 51: CALL FC21 UNIT 02 LASER POWER - $A_DBB[514] / READ TOOL NUMBER MONITOR SPINDLES STA 01R IN CNC
   // $A_DBB[18] IN CNC
   RUNG wire#powerrail
      "LBP_TransferSelData"(Enable := "M_ONE", Funct := #READ, IVAR1 := "DB2400_DBB_VALUES".DBB_DBW_DBD_VAL_514, IVAR2 := -1, S7Var := "DB2401_DBB_DEFINE".DBW_514, Error => #ERROR, ErrCode => #ERROR_CODE)
   END_RUNG
   // the same network as SCL:
   "LBP_TransferSelData"(Enable := "M_ONE",
                         Funct := #READ,
                         IVAR1 := "DB2400_DBB_VALUES".DBB_DBW_DBD_VAL_514,
                         IVAR2 := -1,
                         S7Var := "DB2401_DBB_DEFINE".DBW_514,
                         Error => #ERROR,
                         ErrCode => #ERROR_CODE);
END_REGION

REGION Network 52: CALL FC21 UNIT 02 LASER PROCESSING (0=CORE / 1=RING / 3=BRIGHTLINE WELD) ($A_DBB[516]) / READ TOOL NUMBER MONITOR SPINDLES STA 01R IN CNC
   // $A_DBB[18] IN CNC
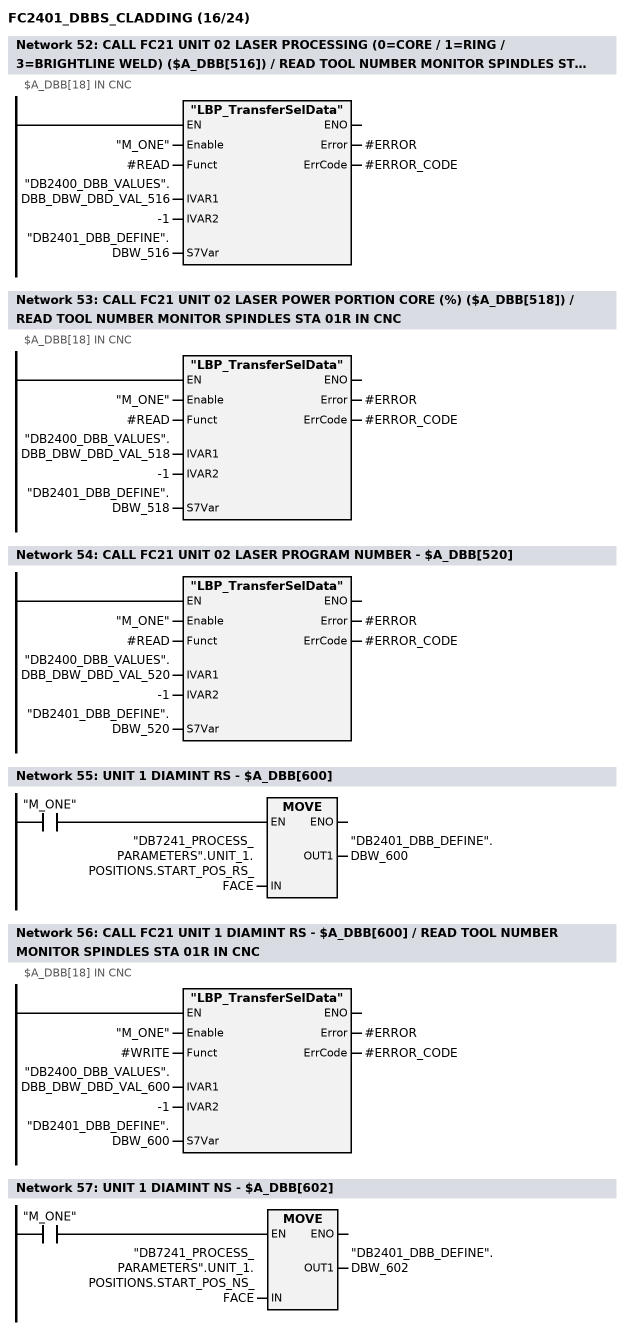
   RUNG wire#powerrail
      "LBP_TransferSelData"(Enable := "M_ONE", Funct := #READ, IVAR1 := "DB2400_DBB_VALUES".DBB_DBW_DBD_VAL_516, IVAR2 := -1, S7Var := "DB2401_DBB_DEFINE".DBW_516, Error => #ERROR, ErrCode => #ERROR_CODE)
   END_RUNG
   // the same network as SCL:
   "LBP_TransferSelData"(Enable := "M_ONE",
                         Funct := #READ,
                         IVAR1 := "DB2400_DBB_VALUES".DBB_DBW_DBD_VAL_516,
                         IVAR2 := -1,
                         S7Var := "DB2401_DBB_DEFINE".DBW_516,
                         Error => #ERROR,
                         ErrCode => #ERROR_CODE);
END_REGION

REGION Network 53: CALL FC21 UNIT 02 LASER POWER PORTION CORE (%) ($A_DBB[518]) / READ TOOL NUMBER MONITOR SPINDLES STA 01R IN CNC
   // $A_DBB[18] IN CNC
   RUNG wire#powerrail
      "LBP_TransferSelData"(Enable := "M_ONE", Funct := #READ, IVAR1 := "DB2400_DBB_VALUES".DBB_DBW_DBD_VAL_518, IVAR2 := -1, S7Var := "DB2401_DBB_DEFINE".DBW_518, Error => #ERROR, ErrCode => #ERROR_CODE)
   END_RUNG
   // the same network as SCL:
   "LBP_TransferSelData"(Enable := "M_ONE",
                         Funct := #READ,
                         IVAR1 := "DB2400_DBB_VALUES".DBB_DBW_DBD_VAL_518,
                         IVAR2 := -1,
                         S7Var := "DB2401_DBB_DEFINE".DBW_518,
                         Error => #ERROR,
                         ErrCode => #ERROR_CODE);
END_REGION

REGION Network 54: CALL FC21 UNIT 02 LASER PROGRAM NUMBER - $A_DBB[520]
   RUNG wire#powerrail
      "LBP_TransferSelData"(Enable := "M_ONE", Funct := #READ, IVAR1 := "DB2400_DBB_VALUES".DBB_DBW_DBD_VAL_520, IVAR2 := -1, S7Var := "DB2401_DBB_DEFINE".DBW_520, Error => #ERROR, ErrCode => #ERROR_CODE)
   END_RUNG
   // the same network as SCL:
   "LBP_TransferSelData"(Enable := "M_ONE",
                         Funct := #READ,
                         IVAR1 := "DB2400_DBB_VALUES".DBB_DBW_DBD_VAL_520,
                         IVAR2 := -1,
                         S7Var := "DB2401_DBB_DEFINE".DBW_520,
                         Error => #ERROR,
                         ErrCode => #ERROR_CODE);
END_REGION

REGION Network 55: UNIT 1 DIAMINT RS - $A_DBB[600]
   RUNG wire#powerrail
      Contact( "M_ONE" )
      Move(in := "DB7241_PROCESS_PARAMETERS".UNIT_1.POSITIONS.START_POS_RS_FACE, out1 => "DB2401_DBB_DEFINE".DBW_600)
   END_RUNG
   // the same network as SCL:
   IF "M_ONE" THEN
       "DB2401_DBB_DEFINE".DBW_600 := "DB7241_PROCESS_PARAMETERS".UNIT_1.POSITIONS.START_POS_RS_FACE;
   END_IF;
END_REGION

REGION Network 56: CALL FC21 UNIT 1 DIAMINT RS - $A_DBB[600] / READ TOOL NUMBER MONITOR SPINDLES STA 01R IN CNC
   // $A_DBB[18] IN CNC
   RUNG wire#powerrail
      "LBP_TransferSelData"(Enable := "M_ONE", Funct := #WRITE, IVAR1 := "DB2400_DBB_VALUES".DBB_DBW_DBD_VAL_600, IVAR2 := -1, S7Var := "DB2401_DBB_DEFINE".DBW_600, Error => #ERROR, ErrCode => #ERROR_CODE)
   END_RUNG
   // the same network as SCL:
   "LBP_TransferSelData"(Enable := "M_ONE",
                         Funct := #WRITE,
                         IVAR1 := "DB2400_DBB_VALUES".DBB_DBW_DBD_VAL_600,
                         IVAR2 := -1,
                         S7Var := "DB2401_DBB_DEFINE".DBW_600,
                         Error => #ERROR,
                         ErrCode => #ERROR_CODE);
END_REGION

REGION Network 57: UNIT 1 DIAMINT NS - $A_DBB[602]
   RUNG wire#powerrail
      Contact( "M_ONE" )
      Move(in := "DB7241_PROCESS_PARAMETERS".UNIT_1.POSITIONS.START_POS_NS_FACE, out1 => "DB2401_DBB_DEFINE".DBW_602)
   END_RUNG
   // the same network as SCL:
   IF "M_ONE" THEN
       "DB2401_DBB_DEFINE".DBW_602 := "DB7241_PROCESS_PARAMETERS".UNIT_1.POSITIONS.START_POS_NS_FACE;
   END_IF;
END_REGION

REGION Network 58: CALL FC21 UNIT 1 DIAMINT NS - $A_DBB[602] / READ TOOL NUMBER MONITOR SPINDLES STA 01R IN CNC
   // $A_DBB[18] IN CNC
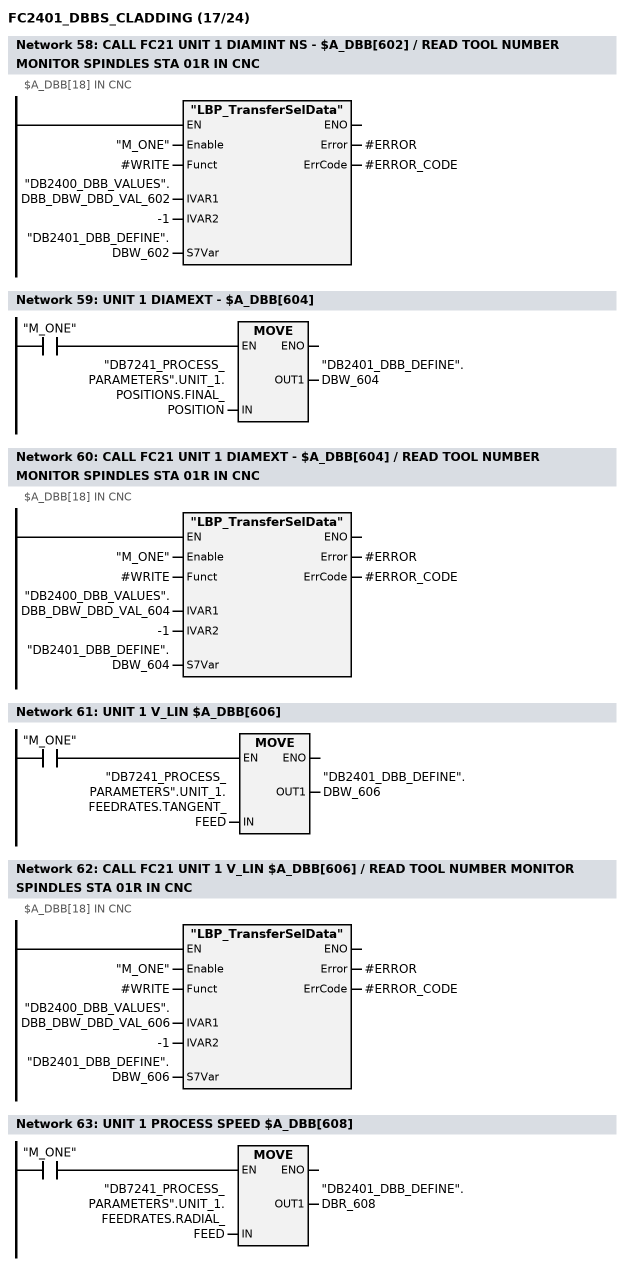
   RUNG wire#powerrail
      "LBP_TransferSelData"(Enable := "M_ONE", Funct := #WRITE, IVAR1 := "DB2400_DBB_VALUES".DBB_DBW_DBD_VAL_602, IVAR2 := -1, S7Var := "DB2401_DBB_DEFINE".DBW_602, Error => #ERROR, ErrCode => #ERROR_CODE)
   END_RUNG
   // the same network as SCL:
   "LBP_TransferSelData"(Enable := "M_ONE",
                         Funct := #WRITE,
                         IVAR1 := "DB2400_DBB_VALUES".DBB_DBW_DBD_VAL_602,
                         IVAR2 := -1,
                         S7Var := "DB2401_DBB_DEFINE".DBW_602,
                         Error => #ERROR,
                         ErrCode => #ERROR_CODE);
END_REGION

REGION Network 59: UNIT 1 DIAMEXT - $A_DBB[604]
   RUNG wire#powerrail
      Contact( "M_ONE" )
      Move(in := "DB7241_PROCESS_PARAMETERS".UNIT_1.POSITIONS.FINAL_POSITION, out1 => "DB2401_DBB_DEFINE".DBW_604)
   END_RUNG
   // the same network as SCL:
   IF "M_ONE" THEN
       "DB2401_DBB_DEFINE".DBW_604 := "DB7241_PROCESS_PARAMETERS".UNIT_1.POSITIONS.FINAL_POSITION;
   END_IF;
END_REGION

REGION Network 60: CALL FC21 UNIT 1 DIAMEXT - $A_DBB[604] / READ TOOL NUMBER MONITOR SPINDLES STA 01R IN CNC
   // $A_DBB[18] IN CNC
   RUNG wire#powerrail
      "LBP_TransferSelData"(Enable := "M_ONE", Funct := #WRITE, IVAR1 := "DB2400_DBB_VALUES".DBB_DBW_DBD_VAL_604, IVAR2 := -1, S7Var := "DB2401_DBB_DEFINE".DBW_604, Error => #ERROR, ErrCode => #ERROR_CODE)
   END_RUNG
   // the same network as SCL:
   "LBP_TransferSelData"(Enable := "M_ONE",
                         Funct := #WRITE,
                         IVAR1 := "DB2400_DBB_VALUES".DBB_DBW_DBD_VAL_604,
                         IVAR2 := -1,
                         S7Var := "DB2401_DBB_DEFINE".DBW_604,
                         Error => #ERROR,
                         ErrCode => #ERROR_CODE);
END_REGION

REGION Network 61: UNIT 1 V_LIN $A_DBB[606]
   RUNG wire#powerrail
      Contact( "M_ONE" )
      Move(in := "DB7241_PROCESS_PARAMETERS".UNIT_1.FEEDRATES.TANGENT_FEED, out1 => "DB2401_DBB_DEFINE".DBW_606)
   END_RUNG
   // the same network as SCL:
   IF "M_ONE" THEN
       "DB2401_DBB_DEFINE".DBW_606 := "DB7241_PROCESS_PARAMETERS".UNIT_1.FEEDRATES.TANGENT_FEED;
   END_IF;
END_REGION

REGION Network 62: CALL FC21 UNIT 1 V_LIN $A_DBB[606] / READ TOOL NUMBER MONITOR SPINDLES STA 01R IN CNC
   // $A_DBB[18] IN CNC
   RUNG wire#powerrail
      "LBP_TransferSelData"(Enable := "M_ONE", Funct := #WRITE, IVAR1 := "DB2400_DBB_VALUES".DBB_DBW_DBD_VAL_606, IVAR2 := -1, S7Var := "DB2401_DBB_DEFINE".DBW_606, Error => #ERROR, ErrCode => #ERROR_CODE)
   END_RUNG
   // the same network as SCL:
   "LBP_TransferSelData"(Enable := "M_ONE",
                         Funct := #WRITE,
                         IVAR1 := "DB2400_DBB_VALUES".DBB_DBW_DBD_VAL_606,
                         IVAR2 := -1,
                         S7Var := "DB2401_DBB_DEFINE".DBW_606,
                         Error => #ERROR,
                         ErrCode => #ERROR_CODE);
END_REGION

REGION Network 63: UNIT 1 PROCESS SPEED $A_DBB[608]
   RUNG wire#powerrail
      Contact( "M_ONE" )
      Move(in := "DB7241_PROCESS_PARAMETERS".UNIT_1.FEEDRATES.RADIAL_FEED, out1 => "DB2401_DBB_DEFINE".DBR_608)
   END_RUNG
   // the same network as SCL:
   IF "M_ONE" THEN
       "DB2401_DBB_DEFINE".DBR_608 := "DB7241_PROCESS_PARAMETERS".UNIT_1.FEEDRATES.RADIAL_FEED;
   END_IF;
END_REGION

REGION Network 64: CALL FC21 UNIT 1 PROCESS SPEED $A_DBB[608] / READ TOOL NUMBER MONITOR SPINDLES STA 01R IN CNC
   // $A_DBB[18] IN CNC
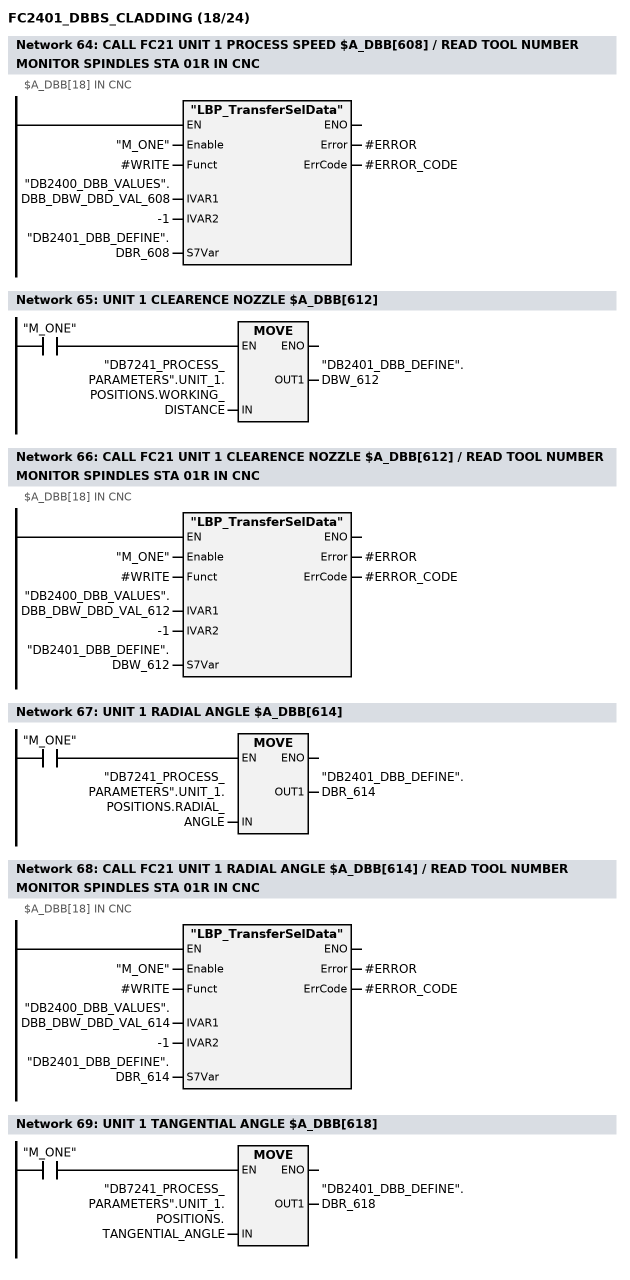
   RUNG wire#powerrail
      "LBP_TransferSelData"(Enable := "M_ONE", Funct := #WRITE, IVAR1 := "DB2400_DBB_VALUES".DBB_DBW_DBD_VAL_608, IVAR2 := -1, S7Var := "DB2401_DBB_DEFINE".DBR_608, Error => #ERROR, ErrCode => #ERROR_CODE)
   END_RUNG
   // the same network as SCL:
   "LBP_TransferSelData"(Enable := "M_ONE",
                         Funct := #WRITE,
                         IVAR1 := "DB2400_DBB_VALUES".DBB_DBW_DBD_VAL_608,
                         IVAR2 := -1,
                         S7Var := "DB2401_DBB_DEFINE".DBR_608,
                         Error => #ERROR,
                         ErrCode => #ERROR_CODE);
END_REGION

REGION Network 65: UNIT 1 CLEARENCE NOZZLE $A_DBB[612]
   RUNG wire#powerrail
      Contact( "M_ONE" )
      Move(in := "DB7241_PROCESS_PARAMETERS".UNIT_1.POSITIONS.WORKING_DISTANCE, out1 => "DB2401_DBB_DEFINE".DBW_612)
   END_RUNG
   // the same network as SCL:
   IF "M_ONE" THEN
       "DB2401_DBB_DEFINE".DBW_612 := "DB7241_PROCESS_PARAMETERS".UNIT_1.POSITIONS.WORKING_DISTANCE;
   END_IF;
END_REGION

REGION Network 66: CALL FC21 UNIT 1 CLEARENCE NOZZLE $A_DBB[612] / READ TOOL NUMBER MONITOR SPINDLES STA 01R IN CNC
   // $A_DBB[18] IN CNC
   RUNG wire#powerrail
      "LBP_TransferSelData"(Enable := "M_ONE", Funct := #WRITE, IVAR1 := "DB2400_DBB_VALUES".DBB_DBW_DBD_VAL_612, IVAR2 := -1, S7Var := "DB2401_DBB_DEFINE".DBW_612, Error => #ERROR, ErrCode => #ERROR_CODE)
   END_RUNG
   // the same network as SCL:
   "LBP_TransferSelData"(Enable := "M_ONE",
                         Funct := #WRITE,
                         IVAR1 := "DB2400_DBB_VALUES".DBB_DBW_DBD_VAL_612,
                         IVAR2 := -1,
                         S7Var := "DB2401_DBB_DEFINE".DBW_612,
                         Error => #ERROR,
                         ErrCode => #ERROR_CODE);
END_REGION

REGION Network 67: UNIT 1 RADIAL ANGLE $A_DBB[614]
   RUNG wire#powerrail
      Contact( "M_ONE" )
      Move(in := "DB7241_PROCESS_PARAMETERS".UNIT_1.POSITIONS.RADIAL_ANGLE, out1 => "DB2401_DBB_DEFINE".DBR_614)
   END_RUNG
   // the same network as SCL:
   IF "M_ONE" THEN
       "DB2401_DBB_DEFINE".DBR_614 := "DB7241_PROCESS_PARAMETERS".UNIT_1.POSITIONS.RADIAL_ANGLE;
   END_IF;
END_REGION

REGION Network 68: CALL FC21 UNIT 1 RADIAL ANGLE $A_DBB[614] / READ TOOL NUMBER MONITOR SPINDLES STA 01R IN CNC
   // $A_DBB[18] IN CNC
   RUNG wire#powerrail
      "LBP_TransferSelData"(Enable := "M_ONE", Funct := #WRITE, IVAR1 := "DB2400_DBB_VALUES".DBB_DBW_DBD_VAL_614, IVAR2 := -1, S7Var := "DB2401_DBB_DEFINE".DBR_614, Error => #ERROR, ErrCode => #ERROR_CODE)
   END_RUNG
   // the same network as SCL:
   "LBP_TransferSelData"(Enable := "M_ONE",
                         Funct := #WRITE,
                         IVAR1 := "DB2400_DBB_VALUES".DBB_DBW_DBD_VAL_614,
                         IVAR2 := -1,
                         S7Var := "DB2401_DBB_DEFINE".DBR_614,
                         Error => #ERROR,
                         ErrCode => #ERROR_CODE);
END_REGION

REGION Network 69: UNIT 1 TANGENTIAL ANGLE $A_DBB[618]
   RUNG wire#powerrail
      Contact( "M_ONE" )
      Move(in := "DB7241_PROCESS_PARAMETERS".UNIT_1.POSITIONS.TANGENTIAL_ANGLE, out1 => "DB2401_DBB_DEFINE".DBR_618)
   END_RUNG
   // the same network as SCL:
   IF "M_ONE" THEN
       "DB2401_DBB_DEFINE".DBR_618 := "DB7241_PROCESS_PARAMETERS".UNIT_1.POSITIONS.TANGENTIAL_ANGLE;
   END_IF;
END_REGION

REGION Network 70: CALL FC21 UNIT 1 TANGENTIAL ANGLE $A_DBB[618] / READ TOOL NUMBER MONITOR SPINDLES STA 01R IN CNC
   // $A_DBB[18] IN CNC
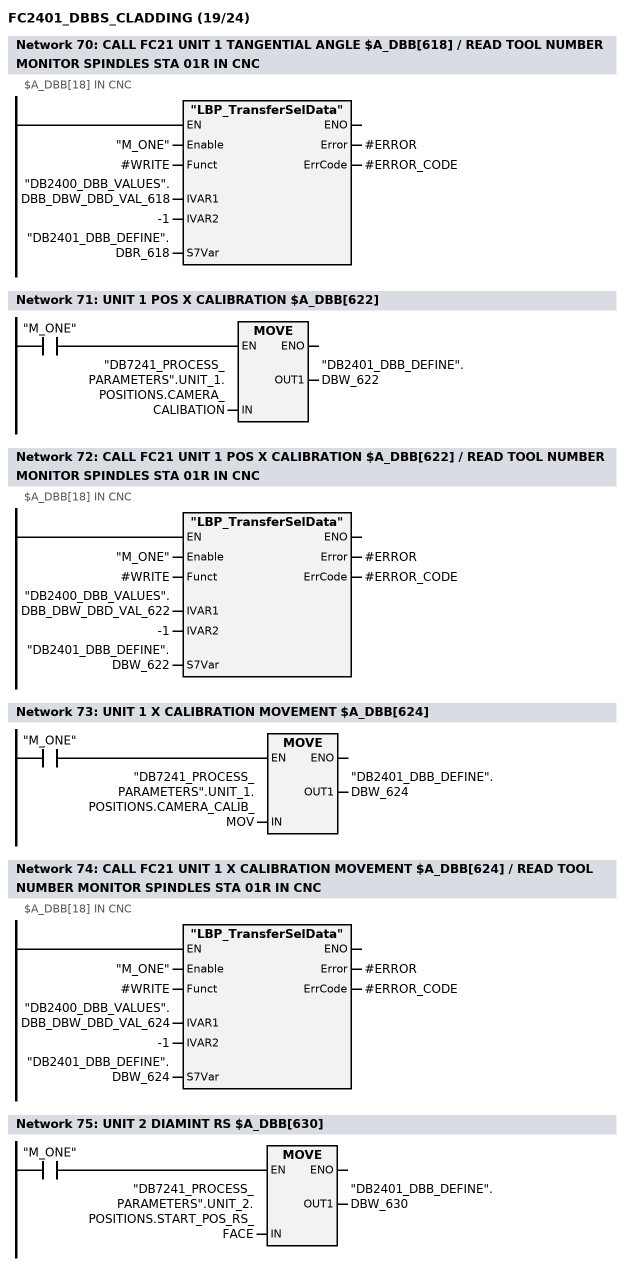
   RUNG wire#powerrail
      "LBP_TransferSelData"(Enable := "M_ONE", Funct := #WRITE, IVAR1 := "DB2400_DBB_VALUES".DBB_DBW_DBD_VAL_618, IVAR2 := -1, S7Var := "DB2401_DBB_DEFINE".DBR_618, Error => #ERROR, ErrCode => #ERROR_CODE)
   END_RUNG
   // the same network as SCL:
   "LBP_TransferSelData"(Enable := "M_ONE",
                         Funct := #WRITE,
                         IVAR1 := "DB2400_DBB_VALUES".DBB_DBW_DBD_VAL_618,
                         IVAR2 := -1,
                         S7Var := "DB2401_DBB_DEFINE".DBR_618,
                         Error => #ERROR,
                         ErrCode => #ERROR_CODE);
END_REGION

REGION Network 71: UNIT 1 POS X CALIBRATION $A_DBB[622]
   RUNG wire#powerrail
      Contact( "M_ONE" )
      Move(in := "DB7241_PROCESS_PARAMETERS".UNIT_1.POSITIONS.CAMERA_CALIBATION, out1 => "DB2401_DBB_DEFINE".DBW_622)
   END_RUNG
   // the same network as SCL:
   IF "M_ONE" THEN
       "DB2401_DBB_DEFINE".DBW_622 := "DB7241_PROCESS_PARAMETERS".UNIT_1.POSITIONS.CAMERA_CALIBATION;
   END_IF;
END_REGION

REGION Network 72: CALL FC21 UNIT 1 POS X CALIBRATION $A_DBB[622] / READ TOOL NUMBER MONITOR SPINDLES STA 01R IN CNC
   // $A_DBB[18] IN CNC
   RUNG wire#powerrail
      "LBP_TransferSelData"(Enable := "M_ONE", Funct := #WRITE, IVAR1 := "DB2400_DBB_VALUES".DBB_DBW_DBD_VAL_622, IVAR2 := -1, S7Var := "DB2401_DBB_DEFINE".DBW_622, Error => #ERROR, ErrCode => #ERROR_CODE)
   END_RUNG
   // the same network as SCL:
   "LBP_TransferSelData"(Enable := "M_ONE",
                         Funct := #WRITE,
                         IVAR1 := "DB2400_DBB_VALUES".DBB_DBW_DBD_VAL_622,
                         IVAR2 := -1,
                         S7Var := "DB2401_DBB_DEFINE".DBW_622,
                         Error => #ERROR,
                         ErrCode => #ERROR_CODE);
END_REGION

REGION Network 73: UNIT 1 X CALIBRATION MOVEMENT $A_DBB[624]
   RUNG wire#powerrail
      Contact( "M_ONE" )
      Move(in := "DB7241_PROCESS_PARAMETERS".UNIT_1.POSITIONS.CAMERA_CALIB_MOV, out1 => "DB2401_DBB_DEFINE".DBW_624)
   END_RUNG
   // the same network as SCL:
   IF "M_ONE" THEN
       "DB2401_DBB_DEFINE".DBW_624 := "DB7241_PROCESS_PARAMETERS".UNIT_1.POSITIONS.CAMERA_CALIB_MOV;
   END_IF;
END_REGION

REGION Network 74: CALL FC21 UNIT 1 X CALIBRATION MOVEMENT $A_DBB[624] / READ TOOL NUMBER MONITOR SPINDLES STA 01R IN CNC
   // $A_DBB[18] IN CNC
   RUNG wire#powerrail
      "LBP_TransferSelData"(Enable := "M_ONE", Funct := #WRITE, IVAR1 := "DB2400_DBB_VALUES".DBB_DBW_DBD_VAL_624, IVAR2 := -1, S7Var := "DB2401_DBB_DEFINE".DBW_624, Error => #ERROR, ErrCode => #ERROR_CODE)
   END_RUNG
   // the same network as SCL:
   "LBP_TransferSelData"(Enable := "M_ONE",
                         Funct := #WRITE,
                         IVAR1 := "DB2400_DBB_VALUES".DBB_DBW_DBD_VAL_624,
                         IVAR2 := -1,
                         S7Var := "DB2401_DBB_DEFINE".DBW_624,
                         Error => #ERROR,
                         ErrCode => #ERROR_CODE);
END_REGION

REGION Network 75: UNIT 2 DIAMINT RS $A_DBB[630]
   RUNG wire#powerrail
      Contact( "M_ONE" )
      Move(in := "DB7241_PROCESS_PARAMETERS".UNIT_2.POSITIONS.START_POS_RS_FACE, out1 => "DB2401_DBB_DEFINE".DBW_630)
   END_RUNG
   // the same network as SCL:
   IF "M_ONE" THEN
       "DB2401_DBB_DEFINE".DBW_630 := "DB7241_PROCESS_PARAMETERS".UNIT_2.POSITIONS.START_POS_RS_FACE;
   END_IF;
END_REGION

REGION Network 76: CALL FC21 UNIT 2 DIAMINT RS $A_DBB[630] / READ TOOL NUMBER MONITOR SPINDLES STA 01R IN CNC
   // $A_DBB[18] IN CNC
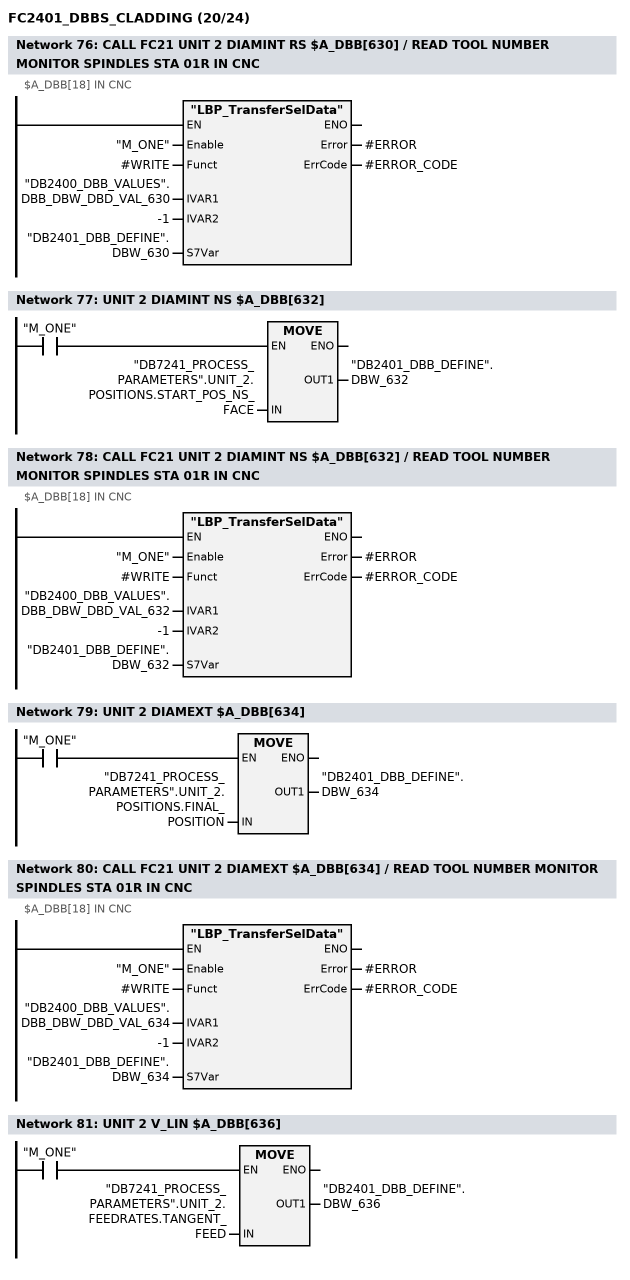
   RUNG wire#powerrail
      "LBP_TransferSelData"(Enable := "M_ONE", Funct := #WRITE, IVAR1 := "DB2400_DBB_VALUES".DBB_DBW_DBD_VAL_630, IVAR2 := -1, S7Var := "DB2401_DBB_DEFINE".DBW_630, Error => #ERROR, ErrCode => #ERROR_CODE)
   END_RUNG
   // the same network as SCL:
   "LBP_TransferSelData"(Enable := "M_ONE",
                         Funct := #WRITE,
                         IVAR1 := "DB2400_DBB_VALUES".DBB_DBW_DBD_VAL_630,
                         IVAR2 := -1,
                         S7Var := "DB2401_DBB_DEFINE".DBW_630,
                         Error => #ERROR,
                         ErrCode => #ERROR_CODE);
END_REGION

REGION Network 77: UNIT 2 DIAMINT NS $A_DBB[632]
   RUNG wire#powerrail
      Contact( "M_ONE" )
      Move(in := "DB7241_PROCESS_PARAMETERS".UNIT_2.POSITIONS.START_POS_NS_FACE, out1 => "DB2401_DBB_DEFINE".DBW_632)
   END_RUNG
   // the same network as SCL:
   IF "M_ONE" THEN
       "DB2401_DBB_DEFINE".DBW_632 := "DB7241_PROCESS_PARAMETERS".UNIT_2.POSITIONS.START_POS_NS_FACE;
   END_IF;
END_REGION

REGION Network 78: CALL FC21 UNIT 2 DIAMINT NS $A_DBB[632] / READ TOOL NUMBER MONITOR SPINDLES STA 01R IN CNC
   // $A_DBB[18] IN CNC
   RUNG wire#powerrail
      "LBP_TransferSelData"(Enable := "M_ONE", Funct := #WRITE, IVAR1 := "DB2400_DBB_VALUES".DBB_DBW_DBD_VAL_632, IVAR2 := -1, S7Var := "DB2401_DBB_DEFINE".DBW_632, Error => #ERROR, ErrCode => #ERROR_CODE)
   END_RUNG
   // the same network as SCL:
   "LBP_TransferSelData"(Enable := "M_ONE",
                         Funct := #WRITE,
                         IVAR1 := "DB2400_DBB_VALUES".DBB_DBW_DBD_VAL_632,
                         IVAR2 := -1,
                         S7Var := "DB2401_DBB_DEFINE".DBW_632,
                         Error => #ERROR,
                         ErrCode => #ERROR_CODE);
END_REGION

REGION Network 79: UNIT 2 DIAMEXT $A_DBB[634]
   RUNG wire#powerrail
      Contact( "M_ONE" )
      Move(in := "DB7241_PROCESS_PARAMETERS".UNIT_2.POSITIONS.FINAL_POSITION, out1 => "DB2401_DBB_DEFINE".DBW_634)
   END_RUNG
   // the same network as SCL:
   IF "M_ONE" THEN
       "DB2401_DBB_DEFINE".DBW_634 := "DB7241_PROCESS_PARAMETERS".UNIT_2.POSITIONS.FINAL_POSITION;
   END_IF;
END_REGION

REGION Network 80: CALL FC21 UNIT 2 DIAMEXT $A_DBB[634] / READ TOOL NUMBER MONITOR SPINDLES STA 01R IN CNC
   // $A_DBB[18] IN CNC
   RUNG wire#powerrail
      "LBP_TransferSelData"(Enable := "M_ONE", Funct := #WRITE, IVAR1 := "DB2400_DBB_VALUES".DBB_DBW_DBD_VAL_634, IVAR2 := -1, S7Var := "DB2401_DBB_DEFINE".DBW_634, Error => #ERROR, ErrCode => #ERROR_CODE)
   END_RUNG
   // the same network as SCL:
   "LBP_TransferSelData"(Enable := "M_ONE",
                         Funct := #WRITE,
                         IVAR1 := "DB2400_DBB_VALUES".DBB_DBW_DBD_VAL_634,
                         IVAR2 := -1,
                         S7Var := "DB2401_DBB_DEFINE".DBW_634,
                         Error => #ERROR,
                         ErrCode => #ERROR_CODE);
END_REGION

REGION Network 81: UNIT 2 V_LIN $A_DBB[636]
   RUNG wire#powerrail
      Contact( "M_ONE" )
      Move(in := "DB7241_PROCESS_PARAMETERS".UNIT_2.FEEDRATES.TANGENT_FEED, out1 => "DB2401_DBB_DEFINE".DBW_636)
   END_RUNG
   // the same network as SCL:
   IF "M_ONE" THEN
       "DB2401_DBB_DEFINE".DBW_636 := "DB7241_PROCESS_PARAMETERS".UNIT_2.FEEDRATES.TANGENT_FEED;
   END_IF;
END_REGION

REGION Network 82: CALL FC21 UNIT 2 V_LIN $A_DBB[636] / READ TOOL NUMBER MONITOR SPINDLES STA 01R IN CNC
   // $A_DBB[18] IN CNC
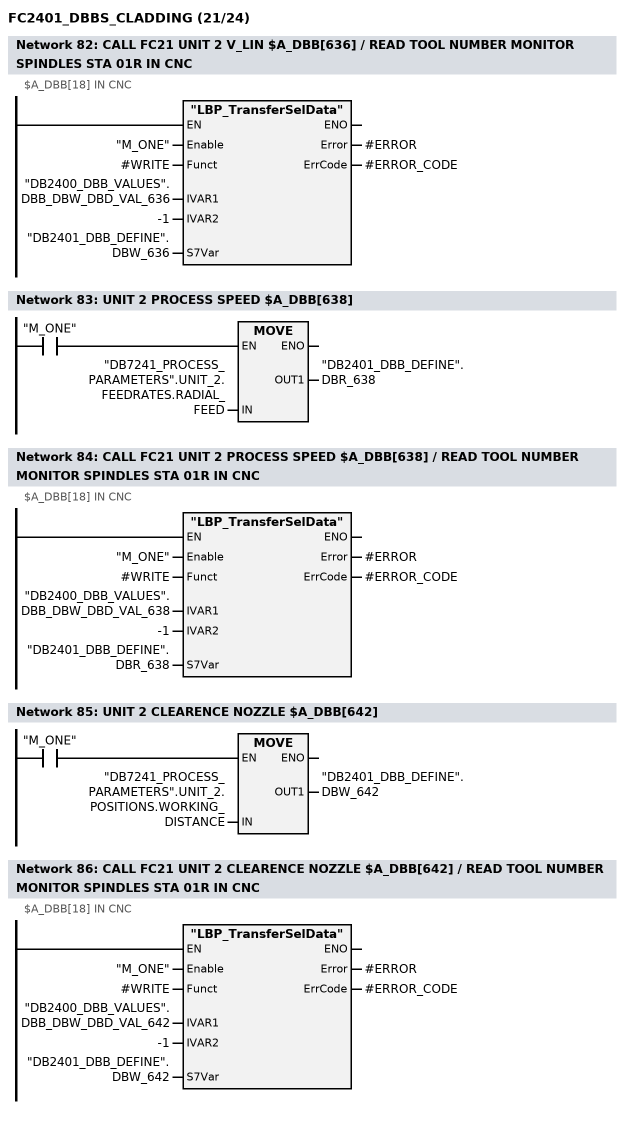
   RUNG wire#powerrail
      "LBP_TransferSelData"(Enable := "M_ONE", Funct := #WRITE, IVAR1 := "DB2400_DBB_VALUES".DBB_DBW_DBD_VAL_636, IVAR2 := -1, S7Var := "DB2401_DBB_DEFINE".DBW_636, Error => #ERROR, ErrCode => #ERROR_CODE)
   END_RUNG
   // the same network as SCL:
   "LBP_TransferSelData"(Enable := "M_ONE",
                         Funct := #WRITE,
                         IVAR1 := "DB2400_DBB_VALUES".DBB_DBW_DBD_VAL_636,
                         IVAR2 := -1,
                         S7Var := "DB2401_DBB_DEFINE".DBW_636,
                         Error => #ERROR,
                         ErrCode => #ERROR_CODE);
END_REGION

REGION Network 83: UNIT 2 PROCESS SPEED $A_DBB[638]
   RUNG wire#powerrail
      Contact( "M_ONE" )
      Move(in := "DB7241_PROCESS_PARAMETERS".UNIT_2.FEEDRATES.RADIAL_FEED, out1 => "DB2401_DBB_DEFINE".DBR_638)
   END_RUNG
   // the same network as SCL:
   IF "M_ONE" THEN
       "DB2401_DBB_DEFINE".DBR_638 := "DB7241_PROCESS_PARAMETERS".UNIT_2.FEEDRATES.RADIAL_FEED;
   END_IF;
END_REGION

REGION Network 84: CALL FC21 UNIT 2 PROCESS SPEED $A_DBB[638] / READ TOOL NUMBER MONITOR SPINDLES STA 01R IN CNC
   // $A_DBB[18] IN CNC
   RUNG wire#powerrail
      "LBP_TransferSelData"(Enable := "M_ONE", Funct := #WRITE, IVAR1 := "DB2400_DBB_VALUES".DBB_DBW_DBD_VAL_638, IVAR2 := -1, S7Var := "DB2401_DBB_DEFINE".DBR_638, Error => #ERROR, ErrCode => #ERROR_CODE)
   END_RUNG
   // the same network as SCL:
   "LBP_TransferSelData"(Enable := "M_ONE",
                         Funct := #WRITE,
                         IVAR1 := "DB2400_DBB_VALUES".DBB_DBW_DBD_VAL_638,
                         IVAR2 := -1,
                         S7Var := "DB2401_DBB_DEFINE".DBR_638,
                         Error => #ERROR,
                         ErrCode => #ERROR_CODE);
END_REGION

REGION Network 85: UNIT 2 CLEARENCE NOZZLE $A_DBB[642]
   RUNG wire#powerrail
      Contact( "M_ONE" )
      Move(in := "DB7241_PROCESS_PARAMETERS".UNIT_2.POSITIONS.WORKING_DISTANCE, out1 => "DB2401_DBB_DEFINE".DBW_642)
   END_RUNG
   // the same network as SCL:
   IF "M_ONE" THEN
       "DB2401_DBB_DEFINE".DBW_642 := "DB7241_PROCESS_PARAMETERS".UNIT_2.POSITIONS.WORKING_DISTANCE;
   END_IF;
END_REGION

REGION Network 86: CALL FC21 UNIT 2 CLEARENCE NOZZLE $A_DBB[642] / READ TOOL NUMBER MONITOR SPINDLES STA 01R IN CNC
   // $A_DBB[18] IN CNC
   RUNG wire#powerrail
      "LBP_TransferSelData"(Enable := "M_ONE", Funct := #WRITE, IVAR1 := "DB2400_DBB_VALUES".DBB_DBW_DBD_VAL_642, IVAR2 := -1, S7Var := "DB2401_DBB_DEFINE".DBW_642, Error => #ERROR, ErrCode => #ERROR_CODE)
   END_RUNG
   // the same network as SCL:
   "LBP_TransferSelData"(Enable := "M_ONE",
                         Funct := #WRITE,
                         IVAR1 := "DB2400_DBB_VALUES".DBB_DBW_DBD_VAL_642,
                         IVAR2 := -1,
                         S7Var := "DB2401_DBB_DEFINE".DBW_642,
                         Error => #ERROR,
                         ErrCode => #ERROR_CODE);
END_REGION

REGION Network 87: CALL FC21 UNIT 2 RADIAL ANGLE $A_DBB[644] / READ TOOL NUMBER MONITOR SPINDLES STA 01R IN CNC
   // $A_DBB[18] IN CNC
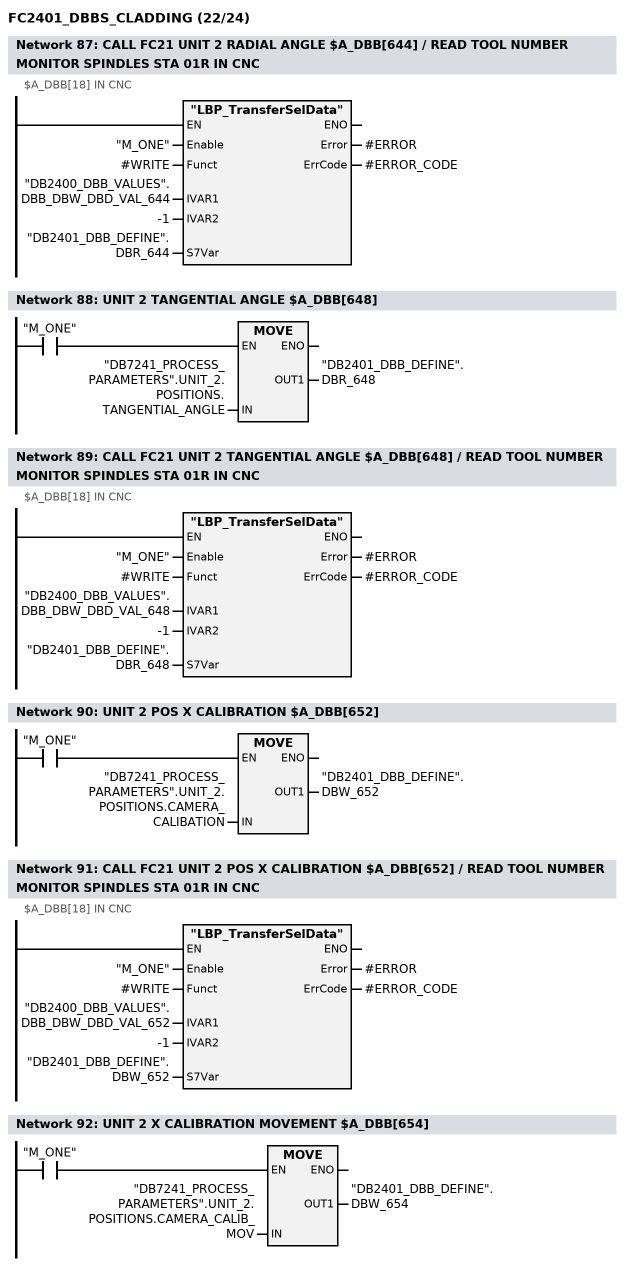
   RUNG wire#powerrail
      "LBP_TransferSelData"(Enable := "M_ONE", Funct := #WRITE, IVAR1 := "DB2400_DBB_VALUES".DBB_DBW_DBD_VAL_644, IVAR2 := -1, S7Var := "DB2401_DBB_DEFINE".DBR_644, Error => #ERROR, ErrCode => #ERROR_CODE)
   END_RUNG
   // the same network as SCL:
   "LBP_TransferSelData"(Enable := "M_ONE",
                         Funct := #WRITE,
                         IVAR1 := "DB2400_DBB_VALUES".DBB_DBW_DBD_VAL_644,
                         IVAR2 := -1,
                         S7Var := "DB2401_DBB_DEFINE".DBR_644,
                         Error => #ERROR,
                         ErrCode => #ERROR_CODE);
END_REGION

REGION Network 88: UNIT 2 TANGENTIAL ANGLE $A_DBB[648]
   RUNG wire#powerrail
      Contact( "M_ONE" )
      Move(in := "DB7241_PROCESS_PARAMETERS".UNIT_2.POSITIONS.TANGENTIAL_ANGLE, out1 => "DB2401_DBB_DEFINE".DBR_648)
   END_RUNG
   // the same network as SCL:
   IF "M_ONE" THEN
       "DB2401_DBB_DEFINE".DBR_648 := "DB7241_PROCESS_PARAMETERS".UNIT_2.POSITIONS.TANGENTIAL_ANGLE;
   END_IF;
END_REGION

REGION Network 89: CALL FC21 UNIT 2 TANGENTIAL ANGLE $A_DBB[648] / READ TOOL NUMBER MONITOR SPINDLES STA 01R IN CNC
   // $A_DBB[18] IN CNC
   RUNG wire#powerrail
      "LBP_TransferSelData"(Enable := "M_ONE", Funct := #WRITE, IVAR1 := "DB2400_DBB_VALUES".DBB_DBW_DBD_VAL_648, IVAR2 := -1, S7Var := "DB2401_DBB_DEFINE".DBR_648, Error => #ERROR, ErrCode => #ERROR_CODE)
   END_RUNG
   // the same network as SCL:
   "LBP_TransferSelData"(Enable := "M_ONE",
                         Funct := #WRITE,
                         IVAR1 := "DB2400_DBB_VALUES".DBB_DBW_DBD_VAL_648,
                         IVAR2 := -1,
                         S7Var := "DB2401_DBB_DEFINE".DBR_648,
                         Error => #ERROR,
                         ErrCode => #ERROR_CODE);
END_REGION

REGION Network 90: UNIT 2 POS X CALIBRATION $A_DBB[652]
   RUNG wire#powerrail
      Contact( "M_ONE" )
      Move(in := "DB7241_PROCESS_PARAMETERS".UNIT_2.POSITIONS.CAMERA_CALIBATION, out1 => "DB2401_DBB_DEFINE".DBW_652)
   END_RUNG
   // the same network as SCL:
   IF "M_ONE" THEN
       "DB2401_DBB_DEFINE".DBW_652 := "DB7241_PROCESS_PARAMETERS".UNIT_2.POSITIONS.CAMERA_CALIBATION;
   END_IF;
END_REGION

REGION Network 91: CALL FC21 UNIT 2 POS X CALIBRATION $A_DBB[652] / READ TOOL NUMBER MONITOR SPINDLES STA 01R IN CNC
   // $A_DBB[18] IN CNC
   RUNG wire#powerrail
      "LBP_TransferSelData"(Enable := "M_ONE", Funct := #WRITE, IVAR1 := "DB2400_DBB_VALUES".DBB_DBW_DBD_VAL_652, IVAR2 := -1, S7Var := "DB2401_DBB_DEFINE".DBW_652, Error => #ERROR, ErrCode => #ERROR_CODE)
   END_RUNG
   // the same network as SCL:
   "LBP_TransferSelData"(Enable := "M_ONE",
                         Funct := #WRITE,
                         IVAR1 := "DB2400_DBB_VALUES".DBB_DBW_DBD_VAL_652,
                         IVAR2 := -1,
                         S7Var := "DB2401_DBB_DEFINE".DBW_652,
                         Error => #ERROR,
                         ErrCode => #ERROR_CODE);
END_REGION

REGION Network 92: UNIT 2 X CALIBRATION MOVEMENT $A_DBB[654]
   RUNG wire#powerrail
      Contact( "M_ONE" )
      Move(in := "DB7241_PROCESS_PARAMETERS".UNIT_2.POSITIONS.CAMERA_CALIB_MOV, out1 => "DB2401_DBB_DEFINE".DBW_654)
   END_RUNG
   // the same network as SCL:
   IF "M_ONE" THEN
       "DB2401_DBB_DEFINE".DBW_654 := "DB7241_PROCESS_PARAMETERS".UNIT_2.POSITIONS.CAMERA_CALIB_MOV;
   END_IF;
END_REGION

REGION Network 93: CALL FC21 UNIT 2 X CALIBRATION MOVEMENT $A_DBB[654] / READ TOOL NUMBER MONITOR SPINDLES STA 01R IN CNC
   // $A_DBB[18] IN CNC
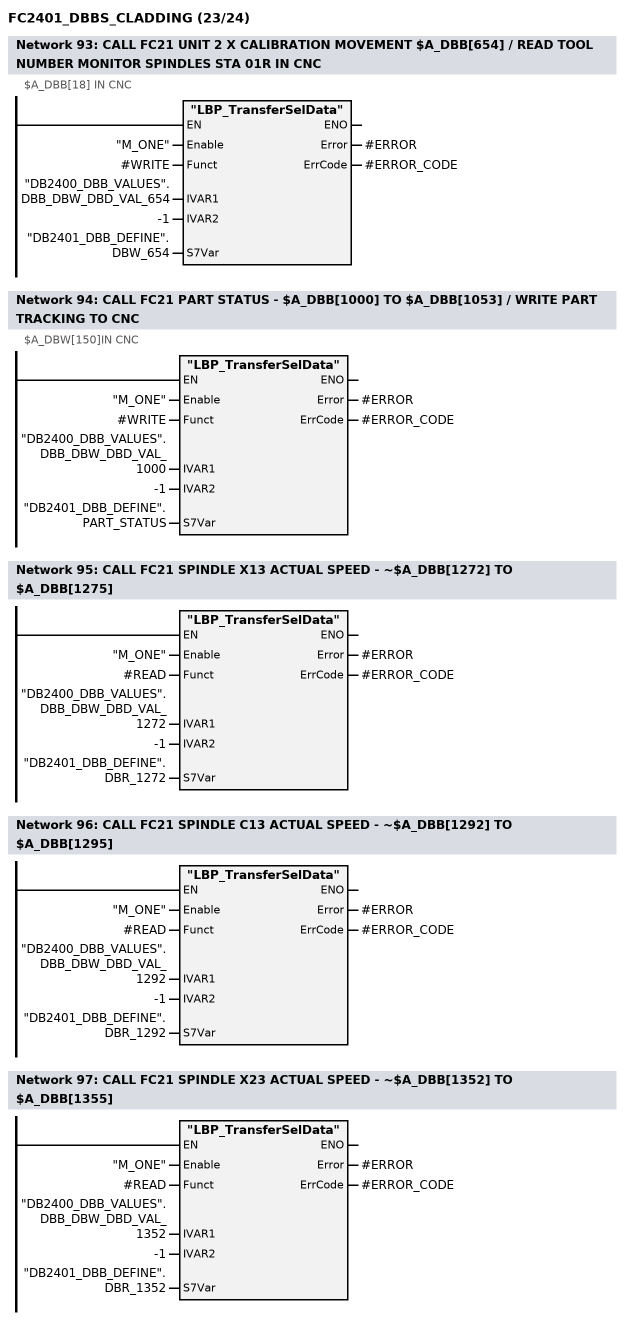
   RUNG wire#powerrail
      "LBP_TransferSelData"(Enable := "M_ONE", Funct := #WRITE, IVAR1 := "DB2400_DBB_VALUES".DBB_DBW_DBD_VAL_654, IVAR2 := -1, S7Var := "DB2401_DBB_DEFINE".DBW_654, Error => #ERROR, ErrCode => #ERROR_CODE)
   END_RUNG
   // the same network as SCL:
   "LBP_TransferSelData"(Enable := "M_ONE",
                         Funct := #WRITE,
                         IVAR1 := "DB2400_DBB_VALUES".DBB_DBW_DBD_VAL_654,
                         IVAR2 := -1,
                         S7Var := "DB2401_DBB_DEFINE".DBW_654,
                         Error => #ERROR,
                         ErrCode => #ERROR_CODE);
END_REGION

REGION Network 94: CALL FC21 PART STATUS - $A_DBB[1000] TO $A_DBB[1053] / WRITE PART TRACKING TO CNC
   // $A_DBW[150]IN CNC
   RUNG wire#powerrail
      "LBP_TransferSelData"(Enable := "M_ONE", Funct := #WRITE, IVAR1 := "DB2400_DBB_VALUES".DBB_DBW_DBD_VAL_1000, IVAR2 := -1, S7Var := "DB2401_DBB_DEFINE".PART_STATUS, Error => #ERROR, ErrCode => #ERROR_CODE)
   END_RUNG
   // the same network as SCL:
   "LBP_TransferSelData"(Enable := "M_ONE",
                         Funct := #WRITE,
                         IVAR1 := "DB2400_DBB_VALUES".DBB_DBW_DBD_VAL_1000,
                         IVAR2 := -1,
                         S7Var := "DB2401_DBB_DEFINE".PART_STATUS,
                         Error => #ERROR,
                         ErrCode => #ERROR_CODE);
END_REGION

REGION Network 95: CALL FC21 SPINDLE X13 ACTUAL SPEED - ~$A_DBB[1272] TO $A_DBB[1275]
   RUNG wire#powerrail
      "LBP_TransferSelData"(Enable := "M_ONE", Funct := #READ, IVAR1 := "DB2400_DBB_VALUES".DBB_DBW_DBD_VAL_1272, IVAR2 := -1, S7Var := "DB2401_DBB_DEFINE".DBR_1272, Error => #ERROR, ErrCode => #ERROR_CODE)
   END_RUNG
   // the same network as SCL:
   "LBP_TransferSelData"(Enable := "M_ONE",
                         Funct := #READ,
                         IVAR1 := "DB2400_DBB_VALUES".DBB_DBW_DBD_VAL_1272,
                         IVAR2 := -1,
                         S7Var := "DB2401_DBB_DEFINE".DBR_1272,
                         Error => #ERROR,
                         ErrCode => #ERROR_CODE);
END_REGION

REGION Network 96: CALL FC21 SPINDLE C13 ACTUAL SPEED - ~$A_DBB[1292] TO $A_DBB[1295]
   RUNG wire#powerrail
      "LBP_TransferSelData"(Enable := "M_ONE", Funct := #READ, IVAR1 := "DB2400_DBB_VALUES".DBB_DBW_DBD_VAL_1292, IVAR2 := -1, S7Var := "DB2401_DBB_DEFINE".DBR_1292, Error => #ERROR, ErrCode => #ERROR_CODE)
   END_RUNG
   // the same network as SCL:
   "LBP_TransferSelData"(Enable := "M_ONE",
                         Funct := #READ,
                         IVAR1 := "DB2400_DBB_VALUES".DBB_DBW_DBD_VAL_1292,
                         IVAR2 := -1,
                         S7Var := "DB2401_DBB_DEFINE".DBR_1292,
                         Error => #ERROR,
                         ErrCode => #ERROR_CODE);
END_REGION

REGION Network 97: CALL FC21 SPINDLE X23 ACTUAL SPEED - ~$A_DBB[1352] TO $A_DBB[1355]
   RUNG wire#powerrail
      "LBP_TransferSelData"(Enable := "M_ONE", Funct := #READ, IVAR1 := "DB2400_DBB_VALUES".DBB_DBW_DBD_VAL_1352, IVAR2 := -1, S7Var := "DB2401_DBB_DEFINE".DBR_1352, Error => #ERROR, ErrCode => #ERROR_CODE)
   END_RUNG
   // the same network as SCL:
   "LBP_TransferSelData"(Enable := "M_ONE",
                         Funct := #READ,
                         IVAR1 := "DB2400_DBB_VALUES".DBB_DBW_DBD_VAL_1352,
                         IVAR2 := -1,
                         S7Var := "DB2401_DBB_DEFINE".DBR_1352,
                         Error => #ERROR,
                         ErrCode => #ERROR_CODE);
END_REGION

REGION Network 98: CALL FC21 SPINDLE C23 ACTUAL SPEED - ~$A_DBB[1372] TO $A_DBB[1375]
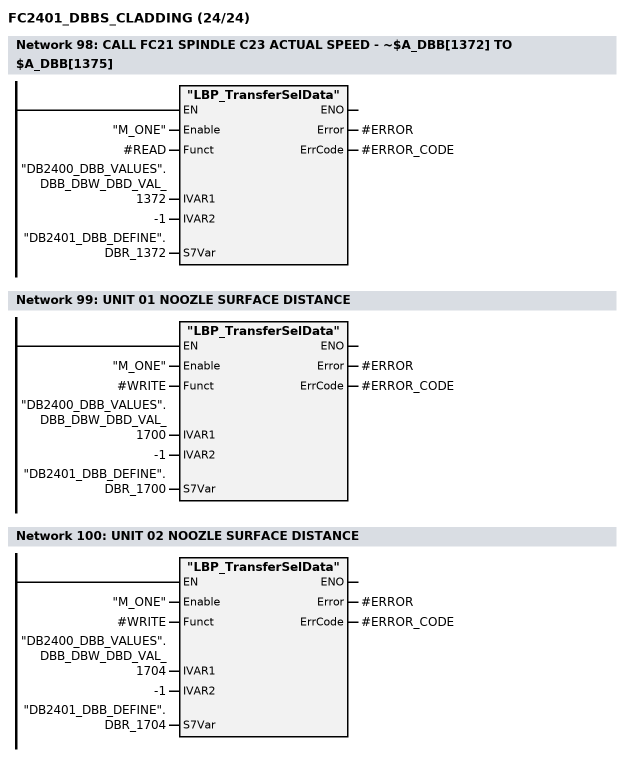
   RUNG wire#powerrail
      "LBP_TransferSelData"(Enable := "M_ONE", Funct := #READ, IVAR1 := "DB2400_DBB_VALUES".DBB_DBW_DBD_VAL_1372, IVAR2 := -1, S7Var := "DB2401_DBB_DEFINE".DBR_1372, Error => #ERROR, ErrCode => #ERROR_CODE)
   END_RUNG
   // the same network as SCL:
   "LBP_TransferSelData"(Enable := "M_ONE",
                         Funct := #READ,
                         IVAR1 := "DB2400_DBB_VALUES".DBB_DBW_DBD_VAL_1372,
                         IVAR2 := -1,
                         S7Var := "DB2401_DBB_DEFINE".DBR_1372,
                         Error => #ERROR,
                         ErrCode => #ERROR_CODE);
END_REGION

REGION Network 99: UNIT 01 NOOZLE SURFACE DISTANCE
   RUNG wire#powerrail
      "LBP_TransferSelData"(Enable := "M_ONE", Funct := #WRITE, IVAR1 := "DB2400_DBB_VALUES".DBB_DBW_DBD_VAL_1700, IVAR2 := -1, S7Var := "DB2401_DBB_DEFINE".DBR_1700, Error => #ERROR, ErrCode => #ERROR_CODE)
   END_RUNG
   // the same network as SCL:
   "LBP_TransferSelData"(Enable := "M_ONE",
                         Funct := #WRITE,
                         IVAR1 := "DB2400_DBB_VALUES".DBB_DBW_DBD_VAL_1700,
                         IVAR2 := -1,
                         S7Var := "DB2401_DBB_DEFINE".DBR_1700,
                         Error => #ERROR,
                         ErrCode => #ERROR_CODE);
END_REGION

REGION Network 100: UNIT 02 NOOZLE SURFACE DISTANCE
   RUNG wire#powerrail
      "LBP_TransferSelData"(Enable := "M_ONE", Funct := #WRITE, IVAR1 := "DB2400_DBB_VALUES".DBB_DBW_DBD_VAL_1704, IVAR2 := -1, S7Var := "DB2401_DBB_DEFINE".DBR_1704, Error => #ERROR, ErrCode => #ERROR_CODE)
   END_RUNG
   // the same network as SCL:
   "LBP_TransferSelData"(Enable := "M_ONE",
                         Funct := #WRITE,
                         IVAR1 := "DB2400_DBB_VALUES".DBB_DBW_DBD_VAL_1704,
                         IVAR2 := -1,
                         S7Var := "DB2401_DBB_DEFINE".DBR_1704,
                         Error => #ERROR,
                         ErrCode => #ERROR_CODE);
END_REGION
END_FUNCTION
